// TIA Portal V20 export
TYPE "LGM_LKinCtrl_Configuration"
// stored: Access Published
   STRUCT
      referenceDesignator { ExternalAccessible := 'False'; ExternalVisible := 'False'; ExternalWritable := 'False'} : WString[25];
      disableAlarms { ExternalAccessible := 'False'; ExternalVisible := 'False'; ExternalWritable := 'False'} : Bool;
      masterControlPopUp { ExternalAccessible := 'False'; ExternalVisible := 'False'; ExternalWritable := 'False'} : Bool;
      groupPower : Struct
         startMode : Array[1.."LKINCTRL_KINEMATICS_AXES"] of DInt;   // startMode of axis; 0: enable NOT position controlled; 1: enable position controlled
         stopMode : Array[1.."LKINCTRL_KINEMATICS_AXES"] of Int;   // stopMode of axis; 0: emergency stop; 1: immediate stop; 2: stop with max dynamics
      END_STRUCT;
      groupHome : Struct
         mode : Array[1.."LKINCTRL_KINEMATICS_AXES"] of Int;   // homing modes for each axis
      END_STRUCT;
      movePath : Struct
         pathDataArray { ExternalAccessible := 'False'; ExternalVisible := 'False'; ExternalWritable := 'False'} : Array[1.."LKINCTRL_NO_OF_PATHS"] of "LKinCtrl_typePathData";
         pointTable { ExternalAccessible := 'False'; ExternalVisible := 'False'; ExternalWritable := 'False'} : Array[1.."LKINCTRL_NO_OF_POINTS_AT_POINT_TABLE"] of "LKinCtrl_typePoint";
         setFlagNames { ExternalAccessible := 'False'; ExternalVisible := 'False'; ExternalWritable := 'False'} : Array[0.."LKINCTRL_NO_OF_LAST_SETFLAG"] of WString;
         valueFlagNames { ExternalAccessible := 'False'; ExternalVisible := 'False'; ExternalWritable := 'False'} : Array[0.."LKINCTRL_NO_OF_LAST_VALUEFLAG"] of WString;
         settings { ExternalAccessible := 'False'; ExternalVisible := 'False'; ExternalWritable := 'False'} : "LKinCtrl_typeSettings";
         pathTransition : DInt;   // initial transition configuration for new path motion (1: use bufferMode and transitionParameter)
         bufferMode : DInt := 1;   // inital bufferMode for new path motion
         transitionParameter : Array[1..5] of LReal;   // initial transitionParameter for new path motion
      END_STRUCT;
   END_STRUCT;
   // groupPower.startMode[1..6] := 1;
   // movePath.pathDataArray[1].pathDataName := 'contour';
   // movePath.pathDataArray[2].pathDataName := 'contourOCS';
   // movePath.pathDataArray[3].pathDataName := 'Packaging';
   // movePath.pathDataArray[4].pathDataName := 'PickAndPlaceTracking';
   // movePath.pathDataArray[5].pathDataName := '- - -';
   // movePath.pathDataArray[1..5].LKinLangInterface.addPointer := 0;
   // movePath.pathDataArray[1..5].LKinLangInterface.retrievePointer := 0;
   // movePath.pathDataArray[1..5].LKinLangInterface.addPointerRestarted := FALSE;
   // movePath.pathDataArray[1..5].LKinLangInterface.ignoreAddPointer := TRUE;
   // movePath.pathDataArray[1..5].LKinLangInterface.bufferLocked := FALSE;
   // movePath.pathDataArray[1..5].LKinLangInterface.preprocessingStop := FALSE;
   // movePath.pathDataArray[1].commands[1..2].cmdType := 1;
   // movePath.pathDataArray[1].commands[3].cmdType := 3;
   // movePath.pathDataArray[1].commands[4..5].cmdType := 1;
   // movePath.pathDataArray[1].commands[6].cmdType := 100;
   // movePath.pathDataArray[1].commands[7].cmdType := 3;
   // movePath.pathDataArray[1].commands[8].cmdType := 1;
   // movePath.pathDataArray[1].commands[9].cmdType := 3;
   // movePath.pathDataArray[1].commands[10].cmdType := 2;
   // movePath.pathDataArray[1].commands[11..20].cmdType := -1;
   // movePath.pathDataArray[2].commands[1].cmdType := 20;
   // movePath.pathDataArray[2].commands[2..3].cmdType := 1;
   // movePath.pathDataArray[2].commands[4].cmdType := 3;
   // movePath.pathDataArray[2].commands[5..6].cmdType := 1;
   // movePath.pathDataArray[2].commands[7].cmdType := 100;
   // movePath.pathDataArray[2].commands[8].cmdType := 3;
   // movePath.pathDataArray[2].commands[9].cmdType := 1;
   // movePath.pathDataArray[2].commands[10].cmdType := 3;
   // movePath.pathDataArray[2].commands[11].cmdType := 2;
   // movePath.pathDataArray[2].commands[12..20].cmdType := -1;
   // movePath.pathDataArray[3].commands[1..6].cmdType := 1;
   // movePath.pathDataArray[3].commands[7..20].cmdType := -1;
   // movePath.pathDataArray[4].commands[1].cmdType := 0;
   // movePath.pathDataArray[4].commands[2].cmdType := 11;
   // movePath.pathDataArray[4].commands[3].cmdType := 100;
   // movePath.pathDataArray[4].commands[4].cmdType := 11;
   // movePath.pathDataArray[4].commands[5].cmdType := 100;
   // movePath.pathDataArray[4].commands[6].cmdType := 11;
   // movePath.pathDataArray[4].commands[7..20].cmdType := -1;
   // movePath.pathDataArray[5].commands[1..20].cmdType := -1;
   // movePath.pathDataArray[1].commands[1..5].cmdActivated := TRUE;
   // movePath.pathDataArray[1].commands[6].cmdActivated := FALSE;
   // movePath.pathDataArray[1].commands[7..20].cmdActivated := TRUE;
   // movePath.pathDataArray[2].commands[1..6].cmdActivated := TRUE;
   // movePath.pathDataArray[2].commands[7].cmdActivated := FALSE;
   // movePath.pathDataArray[2].commands[8..20].cmdActivated := TRUE;
   // movePath.pathDataArray[3].commands[1..20].cmdActivated := TRUE;
   // movePath.pathDataArray[4].commands[1..20].cmdActivated := TRUE;
   // movePath.pathDataArray[5].commands[1..20].cmdActivated := TRUE;
   // movePath.pathDataArray[1].commands[1].cmdName := 'B_up';
   // movePath.pathDataArray[1].commands[2].cmdName := 'B';
   // movePath.pathDataArray[1].commands[3].cmdName := 'Circ';
   // movePath.pathDataArray[1].commands[4].cmdName := 'D_up';
   // movePath.pathDataArray[1].commands[5].cmdName := 'D';
   // movePath.pathDataArray[1].commands[6].cmdName := '';
   // movePath.pathDataArray[1].commands[7].cmdName := 'S_up';
   // movePath.pathDataArray[1].commands[8].cmdName := 'F';
   // movePath.pathDataArray[1].commands[9].cmdName := 'S_lo';
   // movePath.pathDataArray[1].commands[10].cmdName := '- - -';
   // movePath.pathDataArray[1].commands[11].cmdName := '';
   // movePath.pathDataArray[1].commands[12].cmdName := '- - -';
   // movePath.pathDataArray[1].commands[13..20].cmdName := '';
   // movePath.pathDataArray[2].commands[1].cmdName := '';
   // movePath.pathDataArray[2].commands[2].cmdName := 'B_up';
   // movePath.pathDataArray[2].commands[3].cmdName := 'B';
   // movePath.pathDataArray[2].commands[4].cmdName := 'Circ';
   // movePath.pathDataArray[2].commands[5].cmdName := 'D_up';
   // movePath.pathDataArray[2].commands[6].cmdName := 'D';
   // movePath.pathDataArray[2].commands[7].cmdName := '';
   // movePath.pathDataArray[2].commands[8].cmdName := 'S_up';
   // movePath.pathDataArray[2].commands[9].cmdName := 'F';
   // movePath.pathDataArray[2].commands[10].cmdName := 'S_lo';
   // movePath.pathDataArray[2].commands[11].cmdName := '- - -';
   // movePath.pathDataArray[2].commands[12..20].cmdName := '';
   // movePath.pathDataArray[3].commands[1..20].cmdName := '- - -';
   // movePath.pathDataArray[4].commands[1..20].cmdName := '- - -';
   // movePath.pathDataArray[5].commands[1..20].cmdName := '- - -';
   // movePath.pathDataArray[1].commands[1..20].point := -1;
   // movePath.pathDataArray[2].commands[1..20].point := -1;
   // movePath.pathDataArray[3].commands[1..3].point := -1;
   // movePath.pathDataArray[3].commands[4].point := 1;
   // movePath.pathDataArray[3].commands[5].point := 2;
   // movePath.pathDataArray[3].commands[6].point := 1;
   // movePath.pathDataArray[3].commands[7..20].point := -1;
   // movePath.pathDataArray[4].commands[1..20].point := -1;
   // movePath.pathDataArray[5].commands[1..20].point := -1;
   // movePath.pathDataArray[1].commands[1..2].measurementCmd := 0;
   // movePath.pathDataArray[1].commands[3].measurementCmd := 1;
   // movePath.pathDataArray[1].commands[4..20].measurementCmd := 0;
   // movePath.pathDataArray[2].commands[1..20].measurementCmd := 0;
   // movePath.pathDataArray[3].commands[1..20].measurementCmd := 0;
   // movePath.pathDataArray[4].commands[1..20].measurementCmd := 0;
   // movePath.pathDataArray[5].commands[1..20].measurementCmd := 0;
   // movePath.pathDataArray[1].commands[1..3].cmdCoordinates.cartesianPosition.x := 0.0;
   // movePath.pathDataArray[1].commands[4..5].cmdCoordinates.cartesianPosition.x := 10.0;
   // movePath.pathDataArray[1].commands[6..7].cmdCoordinates.cartesianPosition.x := 0.0;
   // movePath.pathDataArray[1].commands[8].cmdCoordinates.cartesianPosition.x := 5.74;
   // movePath.pathDataArray[1].commands[9..20].cmdCoordinates.cartesianPosition.x := 0.0;
   // movePath.pathDataArray[2].commands[1].cmdCoordinates.cartesianPosition.x := 100.0;
   // movePath.pathDataArray[2].commands[2..4].cmdCoordinates.cartesianPosition.x := 0.0;
   // movePath.pathDataArray[2].commands[5..6].cmdCoordinates.cartesianPosition.x := 10.0;
   // movePath.pathDataArray[2].commands[7..8].cmdCoordinates.cartesianPosition.x := 0.0;
   // movePath.pathDataArray[2].commands[9].cmdCoordinates.cartesianPosition.x := 5.74;
   // movePath.pathDataArray[2].commands[10..20].cmdCoordinates.cartesianPosition.x := 0.0;
   // movePath.pathDataArray[3].commands[1..20].cmdCoordinates.cartesianPosition.x := 0.0;
   // movePath.pathDataArray[4].commands[1..3].cmdCoordinates.cartesianPosition.x := 0.0;
   // movePath.pathDataArray[4].commands[4].cmdCoordinates.cartesianPosition.x := 50.0;
   // movePath.pathDataArray[4].commands[5].cmdCoordinates.cartesianPosition.x := 0.0;
   // movePath.pathDataArray[4].commands[6].cmdCoordinates.cartesianPosition.x := 50.0;
   // movePath.pathDataArray[4].commands[7..20].cmdCoordinates.cartesianPosition.x := 0.0;
   // movePath.pathDataArray[5].commands[1..20].cmdCoordinates.cartesianPosition.x := 0.0;
   // movePath.pathDataArray[1].commands[1..2].cmdCoordinates.cartesianPosition.y := 28.28;
   // movePath.pathDataArray[1].commands[3].cmdCoordinates.cartesianPosition.y := 0.0;
   // movePath.pathDataArray[1].commands[4..5].cmdCoordinates.cartesianPosition.y := 10.0;
   // movePath.pathDataArray[1].commands[6..7].cmdCoordinates.cartesianPosition.y := 0.0;
   // movePath.pathDataArray[1].commands[8].cmdCoordinates.cartesianPosition.y := -1.81;
   // movePath.pathDataArray[1].commands[9..20].cmdCoordinates.cartesianPosition.y := 0.0;
   // movePath.pathDataArray[2].commands[1].cmdCoordinates.cartesianPosition.y := 0.0;
   // movePath.pathDataArray[2].commands[2..3].cmdCoordinates.cartesianPosition.y := 28.28;
   // movePath.pathDataArray[2].commands[4].cmdCoordinates.cartesianPosition.y := 0.0;
   // movePath.pathDataArray[2].commands[5..6].cmdCoordinates.cartesianPosition.y := 10.0;
   // movePath.pathDataArray[2].commands[7..8].cmdCoordinates.cartesianPosition.y := 0.0;
   // movePath.pathDataArray[2].commands[9].cmdCoordinates.cartesianPosition.y := -1.81;
   // movePath.pathDataArray[2].commands[10..20].cmdCoordinates.cartesianPosition.y := 0.0;
   // movePath.pathDataArray[3].commands[1..20].cmdCoordinates.cartesianPosition.y := 0.0;
   // movePath.pathDataArray[4].commands[1..20].cmdCoordinates.cartesianPosition.y := 0.0;
   // movePath.pathDataArray[5].commands[1..20].cmdCoordinates.cartesianPosition.y := 0.0;
   // movePath.pathDataArray[1].commands[1].cmdCoordinates.cartesianPosition.z := 50.0;
   // movePath.pathDataArray[1].commands[2..3].cmdCoordinates.cartesianPosition.z := 0.0;
   // movePath.pathDataArray[1].commands[4].cmdCoordinates.cartesianPosition.z := 50.0;
   // movePath.pathDataArray[1].commands[5..9].cmdCoordinates.cartesianPosition.z := 0.0;
   // movePath.pathDataArray[1].commands[10].cmdCoordinates.cartesianPosition.z := 50.0;
   // movePath.pathDataArray[1].commands[11..20].cmdCoordinates.cartesianPosition.z := 0.0;
   // movePath.pathDataArray[2].commands[1].cmdCoordinates.cartesianPosition.z := 0.0;
   // movePath.pathDataArray[2].commands[2].cmdCoordinates.cartesianPosition.z := 50.0;
   // movePath.pathDataArray[2].commands[3..4].cmdCoordinates.cartesianPosition.z := 0.0;
   // movePath.pathDataArray[2].commands[5].cmdCoordinates.cartesianPosition.z := 50.0;
   // movePath.pathDataArray[2].commands[6..10].cmdCoordinates.cartesianPosition.z := 0.0;
   // movePath.pathDataArray[2].commands[11].cmdCoordinates.cartesianPosition.z := 50.0;
   // movePath.pathDataArray[2].commands[12..20].cmdCoordinates.cartesianPosition.z := 0.0;
   // movePath.pathDataArray[3].commands[1].cmdCoordinates.cartesianPosition.z := 50.0;
   // movePath.pathDataArray[3].commands[2].cmdCoordinates.cartesianPosition.z := 10.0;
   // movePath.pathDataArray[3].commands[3].cmdCoordinates.cartesianPosition.z := 50.0;
   // movePath.pathDataArray[3].commands[4..20].cmdCoordinates.cartesianPosition.z := 0.0;
   // movePath.pathDataArray[4].commands[1].cmdCoordinates.cartesianPosition.z := 0.0;
   // movePath.pathDataArray[4].commands[2].cmdCoordinates.cartesianPosition.z := 10.0;
   // movePath.pathDataArray[4].commands[3].cmdCoordinates.cartesianPosition.z := 0.0;
   // movePath.pathDataArray[4].commands[4].cmdCoordinates.cartesianPosition.z := 10.0;
   // movePath.pathDataArray[4].commands[5].cmdCoordinates.cartesianPosition.z := 0.0;
   // movePath.pathDataArray[4].commands[6].cmdCoordinates.cartesianPosition.z := 80.0;
   // movePath.pathDataArray[4].commands[7..20].cmdCoordinates.cartesianPosition.z := 0.0;
   // movePath.pathDataArray[5].commands[1..20].cmdCoordinates.cartesianPosition.z := 0.0;
   // movePath.pathDataArray[1].commands[1..20].cmdCoordinates.cartesianPosition."a" := 0.0;
   // movePath.pathDataArray[2].commands[1..20].cmdCoordinates.cartesianPosition."a" := 0.0;
   // movePath.pathDataArray[3].commands[1..20].cmdCoordinates.cartesianPosition."a" := 0.0;
   // movePath.pathDataArray[4].commands[1..3].cmdCoordinates.cartesianPosition."a" := 0.0;
   // movePath.pathDataArray[4].commands[4].cmdCoordinates.cartesianPosition."a" := 90.0;
   // movePath.pathDataArray[4].commands[5..20].cmdCoordinates.cartesianPosition."a" := 0.0;
   // movePath.pathDataArray[5].commands[1..20].cmdCoordinates.cartesianPosition."a" := 0.0;
   // movePath.pathDataArray[1].commands[1..20].cmdCoordinates.cartesianPosition."b" := 0.0;
   // movePath.pathDataArray[2].commands[1..20].cmdCoordinates.cartesianPosition."b" := 0.0;
   // movePath.pathDataArray[3].commands[1..20].cmdCoordinates.cartesianPosition."b" := 0.0;
   // movePath.pathDataArray[4].commands[1..20].cmdCoordinates.cartesianPosition."b" := 0.0;
   // movePath.pathDataArray[5].commands[1..20].cmdCoordinates.cartesianPosition."b" := 0.0;
   // movePath.pathDataArray[1].commands[1..20].cmdCoordinates.cartesianPosition.c := 0.0;
   // movePath.pathDataArray[2].commands[1..20].cmdCoordinates.cartesianPosition.c := 0.0;
   // movePath.pathDataArray[3].commands[1..20].cmdCoordinates.cartesianPosition.c := 0.0;
   // movePath.pathDataArray[4].commands[1..20].cmdCoordinates.cartesianPosition.c := 0.0;
   // movePath.pathDataArray[5].commands[1..20].cmdCoordinates.cartesianPosition.c := 0.0;
   // movePath.pathDataArray[1].commands[1..20].cmdCoordinates.coordSystem := 0;
   // movePath.pathDataArray[2].commands[1..6].cmdCoordinates.coordSystem := 3;
   // movePath.pathDataArray[2].commands[7].cmdCoordinates.coordSystem := 0;
   // movePath.pathDataArray[2].commands[8..10].cmdCoordinates.coordSystem := 3;
   // movePath.pathDataArray[2].commands[11..20].cmdCoordinates.coordSystem := 0;
   // movePath.pathDataArray[3].commands[1..20].cmdCoordinates.coordSystem := 0;
   // movePath.pathDataArray[4].commands[1].cmdCoordinates.coordSystem := 0;
   // movePath.pathDataArray[4].commands[2].cmdCoordinates.coordSystem := 1;
   // movePath.pathDataArray[4].commands[3].cmdCoordinates.coordSystem := 0;
   // movePath.pathDataArray[4].commands[4].cmdCoordinates.coordSystem := 2;
   // movePath.pathDataArray[4].commands[5..20].cmdCoordinates.coordSystem := 0;
   // movePath.pathDataArray[5].commands[1..20].cmdCoordinates.coordSystem := 0;
   // movePath.pathDataArray[1].commands[1..2].cmdParameters.pathDynamics.velocity := 300.0;
   // movePath.pathDataArray[1].commands[3].cmdParameters.pathDynamics.velocity := 150.0;
   // movePath.pathDataArray[1].commands[4..5].cmdParameters.pathDynamics.velocity := 300.0;
   // movePath.pathDataArray[1].commands[6].cmdParameters.pathDynamics.velocity := 3000.0;
   // movePath.pathDataArray[1].commands[7].cmdParameters.pathDynamics.velocity := 150.0;
   // movePath.pathDataArray[1].commands[8].cmdParameters.pathDynamics.velocity := 300.0;
   // movePath.pathDataArray[1].commands[9].cmdParameters.pathDynamics.velocity := 150.0;
   // movePath.pathDataArray[1].commands[10..20].cmdParameters.pathDynamics.velocity := -1.0;
   // movePath.pathDataArray[2].commands[1].cmdParameters.pathDynamics.velocity := -1.0;
   // movePath.pathDataArray[2].commands[2..3].cmdParameters.pathDynamics.velocity := 300.0;
   // movePath.pathDataArray[2].commands[4].cmdParameters.pathDynamics.velocity := 150.0;
   // movePath.pathDataArray[2].commands[5..6].cmdParameters.pathDynamics.velocity := 300.0;
   // movePath.pathDataArray[2].commands[7].cmdParameters.pathDynamics.velocity := 3000.0;
   // movePath.pathDataArray[2].commands[8].cmdParameters.pathDynamics.velocity := 150.0;
   // movePath.pathDataArray[2].commands[9].cmdParameters.pathDynamics.velocity := 300.0;
   // movePath.pathDataArray[2].commands[10].cmdParameters.pathDynamics.velocity := 150.0;
   // movePath.pathDataArray[2].commands[11..20].cmdParameters.pathDynamics.velocity := -1.0;
   // movePath.pathDataArray[3].commands[1..20].cmdParameters.pathDynamics.velocity := -1.0;
   // movePath.pathDataArray[4].commands[1].cmdParameters.pathDynamics.velocity := -1.0;
   // movePath.pathDataArray[4].commands[2..6].cmdParameters.pathDynamics.velocity := 200.0;
   // movePath.pathDataArray[4].commands[7..20].cmdParameters.pathDynamics.velocity := -1.0;
   // movePath.pathDataArray[5].commands[1..20].cmdParameters.pathDynamics.velocity := -1.0;
   // movePath.pathDataArray[1].commands[1..20].cmdParameters.pathDynamics.acceleration := -1.0;
   // movePath.pathDataArray[2].commands[1..20].cmdParameters.pathDynamics.acceleration := -1.0;
   // movePath.pathDataArray[3].commands[1..20].cmdParameters.pathDynamics.acceleration := -1.0;
   // movePath.pathDataArray[4].commands[1..20].cmdParameters.pathDynamics.acceleration := -1.0;
   // movePath.pathDataArray[5].commands[1..20].cmdParameters.pathDynamics.acceleration := -1.0;
   // movePath.pathDataArray[1].commands[1..20].cmdParameters.pathDynamics.deceleration := -1.0;
   // movePath.pathDataArray[2].commands[1..20].cmdParameters.pathDynamics.deceleration := -1.0;
   // movePath.pathDataArray[3].commands[1..20].cmdParameters.pathDynamics.deceleration := -1.0;
   // movePath.pathDataArray[4].commands[1..20].cmdParameters.pathDynamics.deceleration := -1.0;
   // movePath.pathDataArray[5].commands[1..20].cmdParameters.pathDynamics.deceleration := -1.0;
   // movePath.pathDataArray[1].commands[1..20].cmdParameters.pathDynamics.jerk := -1.0;
   // movePath.pathDataArray[2].commands[1..20].cmdParameters.pathDynamics.jerk := -1.0;
   // movePath.pathDataArray[3].commands[1..20].cmdParameters.pathDynamics.jerk := -1.0;
   // movePath.pathDataArray[4].commands[1..20].cmdParameters.pathDynamics.jerk := -1.0;
   // movePath.pathDataArray[5].commands[1..20].cmdParameters.pathDynamics.jerk := -1.0;
   // movePath.pathDataArray[1].commands[1..20].cmdParameters.orientationDynamics.velocity := -1.0;
   // movePath.pathDataArray[2].commands[1..20].cmdParameters.orientationDynamics.velocity := -1.0;
   // movePath.pathDataArray[3].commands[1..20].cmdParameters.orientationDynamics.velocity := -1.0;
   // movePath.pathDataArray[4].commands[1..20].cmdParameters.orientationDynamics.velocity := -1.0;
   // movePath.pathDataArray[5].commands[1..20].cmdParameters.orientationDynamics.velocity := -1.0;
   // movePath.pathDataArray[1].commands[1..20].cmdParameters.orientationDynamics.acceleration := -1.0;
   // movePath.pathDataArray[2].commands[1..20].cmdParameters.orientationDynamics.acceleration := -1.0;
   // movePath.pathDataArray[3].commands[1..20].cmdParameters.orientationDynamics.acceleration := -1.0;
   // movePath.pathDataArray[4].commands[1..20].cmdParameters.orientationDynamics.acceleration := -1.0;
   // movePath.pathDataArray[5].commands[1..20].cmdParameters.orientationDynamics.acceleration := -1.0;
   // movePath.pathDataArray[1].commands[1..20].cmdParameters.orientationDynamics.deceleration := -1.0;
   // movePath.pathDataArray[2].commands[1..20].cmdParameters.orientationDynamics.deceleration := -1.0;
   // movePath.pathDataArray[3].commands[1..20].cmdParameters.orientationDynamics.deceleration := -1.0;
   // movePath.pathDataArray[4].commands[1..20].cmdParameters.orientationDynamics.deceleration := -1.0;
   // movePath.pathDataArray[5].commands[1..20].cmdParameters.orientationDynamics.deceleration := -1.0;
   // movePath.pathDataArray[1].commands[1..20].cmdParameters.orientationDynamics.jerk := -1.0;
   // movePath.pathDataArray[2].commands[1..20].cmdParameters.orientationDynamics.jerk := -1.0;
   // movePath.pathDataArray[3].commands[1..20].cmdParameters.orientationDynamics.jerk := -1.0;
   // movePath.pathDataArray[4].commands[1..20].cmdParameters.orientationDynamics.jerk := -1.0;
   // movePath.pathDataArray[5].commands[1..20].cmdParameters.orientationDynamics.jerk := -1.0;
   // movePath.pathDataArray[1].commands[1..20].cmdParameters.orientationDirection := 3;
   // movePath.pathDataArray[2].commands[1..20].cmdParameters.orientationDirection := 3;
   // movePath.pathDataArray[3].commands[1..20].cmdParameters.orientationDirection := 3;
   // movePath.pathDataArray[4].commands[1..20].cmdParameters.orientationDirection := 3;
   // movePath.pathDataArray[5].commands[1..20].cmdParameters.orientationDirection := 3;
   // movePath.pathDataArray[1].commands[1..2].cmdParameters.bufferMode := 2;
   // movePath.pathDataArray[1].commands[3..4].cmdParameters.bufferMode := 1;
   // movePath.pathDataArray[1].commands[5].cmdParameters.bufferMode := 2;
   // movePath.pathDataArray[1].commands[6..7].cmdParameters.bufferMode := 1;
   // movePath.pathDataArray[1].commands[8..9].cmdParameters.bufferMode := 2;
   // movePath.pathDataArray[1].commands[10..20].cmdParameters.bufferMode := 1;
   // movePath.pathDataArray[2].commands[1].cmdParameters.bufferMode := 1;
   // movePath.pathDataArray[2].commands[2..3].cmdParameters.bufferMode := 2;
   // movePath.pathDataArray[2].commands[4..5].cmdParameters.bufferMode := 1;
   // movePath.pathDataArray[2].commands[6].cmdParameters.bufferMode := 2;
   // movePath.pathDataArray[2].commands[7..8].cmdParameters.bufferMode := 1;
   // movePath.pathDataArray[2].commands[9..10].cmdParameters.bufferMode := 2;
   // movePath.pathDataArray[2].commands[11..20].cmdParameters.bufferMode := 1;
   // movePath.pathDataArray[3].commands[1..2].cmdParameters.bufferMode := 5;
   // movePath.pathDataArray[3].commands[3].cmdParameters.bufferMode := 1;
   // movePath.pathDataArray[3].commands[4..5].cmdParameters.bufferMode := 5;
   // movePath.pathDataArray[3].commands[6..20].cmdParameters.bufferMode := 1;
   // movePath.pathDataArray[4].commands[1].cmdParameters.bufferMode := 1;
   // movePath.pathDataArray[4].commands[2].cmdParameters.bufferMode := 5;
   // movePath.pathDataArray[4].commands[3..20].cmdParameters.bufferMode := 1;
   // movePath.pathDataArray[5].commands[1..20].cmdParameters.bufferMode := 1;
   // movePath.pathDataArray[1].commands[1].cmdParameters.transitionParameters[1] := -1.0;
   // movePath.pathDataArray[1].commands[1].cmdParameters.transitionParameters[2..5] := 0.0;
   // movePath.pathDataArray[1].commands[2].cmdParameters.transitionParameters[1] := -1.0;
   // movePath.pathDataArray[1].commands[2].cmdParameters.transitionParameters[2..5] := 0.0;
   // movePath.pathDataArray[1].commands[3].cmdParameters.transitionParameters[1] := -1.0;
   // movePath.pathDataArray[1].commands[3].cmdParameters.transitionParameters[2..5] := 0.0;
   // movePath.pathDataArray[1].commands[4].cmdParameters.transitionParameters[1] := -1.0;
   // movePath.pathDataArray[1].commands[4].cmdParameters.transitionParameters[2..5] := 0.0;
   // movePath.pathDataArray[1].commands[5].cmdParameters.transitionParameters[1] := -1.0;
   // movePath.pathDataArray[1].commands[5].cmdParameters.transitionParameters[2..5] := 0.0;
   // movePath.pathDataArray[1].commands[6].cmdParameters.transitionParameters[1] := -1.0;
   // movePath.pathDataArray[1].commands[6].cmdParameters.transitionParameters[2..5] := 0.0;
   // movePath.pathDataArray[1].commands[7].cmdParameters.transitionParameters[1] := -1.0;
   // movePath.pathDataArray[1].commands[7].cmdParameters.transitionParameters[2..5] := 0.0;
   // movePath.pathDataArray[1].commands[8].cmdParameters.transitionParameters[1] := -1.0;
   // movePath.pathDataArray[1].commands[8].cmdParameters.transitionParameters[2..5] := 0.0;
   // movePath.pathDataArray[1].commands[9].cmdParameters.transitionParameters[1] := -1.0;
   // movePath.pathDataArray[1].commands[9].cmdParameters.transitionParameters[2..5] := 0.0;
   // movePath.pathDataArray[1].commands[10].cmdParameters.transitionParameters[1] := -1.0;
   // movePath.pathDataArray[1].commands[10].cmdParameters.transitionParameters[2..5] := 0.0;
   // movePath.pathDataArray[1].commands[11].cmdParameters.transitionParameters[1] := -1.0;
   // movePath.pathDataArray[1].commands[11].cmdParameters.transitionParameters[2..5] := 0.0;
   // movePath.pathDataArray[1].commands[12].cmdParameters.transitionParameters[1] := -1.0;
   // movePath.pathDataArray[1].commands[12].cmdParameters.transitionParameters[2..5] := 0.0;
   // movePath.pathDataArray[1].commands[13].cmdParameters.transitionParameters[1] := -1.0;
   // movePath.pathDataArray[1].commands[13].cmdParameters.transitionParameters[2..5] := 0.0;
   // movePath.pathDataArray[1].commands[14].cmdParameters.transitionParameters[1] := -1.0;
   // movePath.pathDataArray[1].commands[14].cmdParameters.transitionParameters[2..5] := 0.0;
   // movePath.pathDataArray[1].commands[15].cmdParameters.transitionParameters[1] := -1.0;
   // movePath.pathDataArray[1].commands[15].cmdParameters.transitionParameters[2..5] := 0.0;
   // movePath.pathDataArray[1].commands[16].cmdParameters.transitionParameters[1] := -1.0;
   // movePath.pathDataArray[1].commands[16].cmdParameters.transitionParameters[2..5] := 0.0;
   // movePath.pathDataArray[1].commands[17].cmdParameters.transitionParameters[1] := -1.0;
   // movePath.pathDataArray[1].commands[17].cmdParameters.transitionParameters[2..5] := 0.0;
   // movePath.pathDataArray[1].commands[18].cmdParameters.transitionParameters[1] := -1.0;
   // movePath.pathDataArray[1].commands[18].cmdParameters.transitionParameters[2..5] := 0.0;
   // movePath.pathDataArray[1].commands[19].cmdParameters.transitionParameters[1] := -1.0;
   // movePath.pathDataArray[1].commands[19].cmdParameters.transitionParameters[2..5] := 0.0;
   // movePath.pathDataArray[1].commands[20].cmdParameters.transitionParameters[1] := -1.0;
   // movePath.pathDataArray[1].commands[20].cmdParameters.transitionParameters[2..5] := 0.0;
   // movePath.pathDataArray[2].commands[1].cmdParameters.transitionParameters[1..5] := 0.0;
   // movePath.pathDataArray[2].commands[2].cmdParameters.transitionParameters[1] := -1.0;
   // movePath.pathDataArray[2].commands[2].cmdParameters.transitionParameters[2..5] := 0.0;
   // movePath.pathDataArray[2].commands[3].cmdParameters.transitionParameters[1] := -1.0;
   // movePath.pathDataArray[2].commands[3].cmdParameters.transitionParameters[2..5] := 0.0;
   // movePath.pathDataArray[2].commands[4].cmdParameters.transitionParameters[1..5] := 0.0;
   // movePath.pathDataArray[2].commands[5].cmdParameters.transitionParameters[1..5] := 0.0;
   // movePath.pathDataArray[2].commands[6].cmdParameters.transitionParameters[1] := -1.0;
   // movePath.pathDataArray[2].commands[6].cmdParameters.transitionParameters[2..5] := 0.0;
   // movePath.pathDataArray[2].commands[7].cmdParameters.transitionParameters[1] := -1.0;
   // movePath.pathDataArray[2].commands[7].cmdParameters.transitionParameters[2..5] := 0.0;
   // movePath.pathDataArray[2].commands[8].cmdParameters.transitionParameters[1..5] := 0.0;
   // movePath.pathDataArray[2].commands[9].cmdParameters.transitionParameters[1] := -1.0;
   // movePath.pathDataArray[2].commands[9].cmdParameters.transitionParameters[2..5] := 0.0;
   // movePath.pathDataArray[2].commands[10].cmdParameters.transitionParameters[1] := -1.0;
   // movePath.pathDataArray[2].commands[10].cmdParameters.transitionParameters[2..5] := 0.0;
   // movePath.pathDataArray[2].commands[11].cmdParameters.transitionParameters[1] := -1.0;
   // movePath.pathDataArray[2].commands[11].cmdParameters.transitionParameters[2..5] := 0.0;
   // movePath.pathDataArray[2].commands[12].cmdParameters.transitionParameters[1] := -1.0;
   // movePath.pathDataArray[2].commands[12].cmdParameters.transitionParameters[2..5] := 0.0;
   // movePath.pathDataArray[2].commands[13].cmdParameters.transitionParameters[1] := -1.0;
   // movePath.pathDataArray[2].commands[13].cmdParameters.transitionParameters[2..5] := 0.0;
   // movePath.pathDataArray[2].commands[14].cmdParameters.transitionParameters[1] := -1.0;
   // movePath.pathDataArray[2].commands[14].cmdParameters.transitionParameters[2..5] := 0.0;
   // movePath.pathDataArray[2].commands[15].cmdParameters.transitionParameters[1] := -1.0;
   // movePath.pathDataArray[2].commands[15].cmdParameters.transitionParameters[2..5] := 0.0;
   // movePath.pathDataArray[2].commands[16].cmdParameters.transitionParameters[1] := -1.0;
   // movePath.pathDataArray[2].commands[16].cmdParameters.transitionParameters[2..5] := 0.0;
   // movePath.pathDataArray[2].commands[17].cmdParameters.transitionParameters[1] := -1.0;
   // movePath.pathDataArray[2].commands[17].cmdParameters.transitionParameters[2..5] := 0.0;
   // movePath.pathDataArray[2].commands[18].cmdParameters.transitionParameters[1] := -1.0;
   // movePath.pathDataArray[2].commands[18].cmdParameters.transitionParameters[2..5] := 0.0;
   // movePath.pathDataArray[2].commands[19].cmdParameters.transitionParameters[1] := -1.0;
   // movePath.pathDataArray[2].commands[19].cmdParameters.transitionParameters[2..5] := 0.0;
   // movePath.pathDataArray[2].commands[20].cmdParameters.transitionParameters[1] := -1.0;
   // movePath.pathDataArray[2].commands[20].cmdParameters.transitionParameters[2..5] := 0.0;
   // movePath.pathDataArray[3].commands[1].cmdParameters.transitionParameters[1] := -1.0;
   // movePath.pathDataArray[3].commands[1].cmdParameters.transitionParameters[2..5] := 0.0;
   // movePath.pathDataArray[3].commands[2].cmdParameters.transitionParameters[1] := -1.0;
   // movePath.pathDataArray[3].commands[2].cmdParameters.transitionParameters[2..5] := 0.0;
   // movePath.pathDataArray[3].commands[3].cmdParameters.transitionParameters[1] := -1.0;
   // movePath.pathDataArray[3].commands[3].cmdParameters.transitionParameters[2..5] := 0.0;
   // movePath.pathDataArray[3].commands[4].cmdParameters.transitionParameters[1] := -1.0;
   // movePath.pathDataArray[3].commands[4].cmdParameters.transitionParameters[2..5] := 0.0;
   // movePath.pathDataArray[3].commands[5].cmdParameters.transitionParameters[1] := -1.0;
   // movePath.pathDataArray[3].commands[5].cmdParameters.transitionParameters[2..5] := 0.0;
   // movePath.pathDataArray[3].commands[6].cmdParameters.transitionParameters[1] := -1.0;
   // movePath.pathDataArray[3].commands[6].cmdParameters.transitionParameters[2..5] := 0.0;
   // movePath.pathDataArray[3].commands[7].cmdParameters.transitionParameters[1] := -1.0;
   // movePath.pathDataArray[3].commands[7].cmdParameters.transitionParameters[2..5] := 0.0;
   // movePath.pathDataArray[3].commands[8].cmdParameters.transitionParameters[1] := -1.0;
   // movePath.pathDataArray[3].commands[8].cmdParameters.transitionParameters[2..5] := 0.0;
   // movePath.pathDataArray[3].commands[9].cmdParameters.transitionParameters[1] := -1.0;
   // movePath.pathDataArray[3].commands[9].cmdParameters.transitionParameters[2..5] := 0.0;
   // movePath.pathDataArray[3].commands[10].cmdParameters.transitionParameters[1] := -1.0;
   // movePath.pathDataArray[3].commands[10].cmdParameters.transitionParameters[2..5] := 0.0;
   // movePath.pathDataArray[3].commands[11].cmdParameters.transitionParameters[1] := -1.0;
   // movePath.pathDataArray[3].commands[11].cmdParameters.transitionParameters[2..5] := 0.0;
   // movePath.pathDataArray[3].commands[12].cmdParameters.transitionParameters[1] := -1.0;
   // movePath.pathDataArray[3].commands[12].cmdParameters.transitionParameters[2..5] := 0.0;
   // movePath.pathDataArray[3].commands[13].cmdParameters.transitionParameters[1] := -1.0;
   // movePath.pathDataArray[3].commands[13].cmdParameters.transitionParameters[2..5] := 0.0;
   // movePath.pathDataArray[3].commands[14].cmdParameters.transitionParameters[1] := -1.0;
   // movePath.pathDataArray[3].commands[14].cmdParameters.transitionParameters[2..5] := 0.0;
   // movePath.pathDataArray[3].commands[15].cmdParameters.transitionParameters[1] := -1.0;
   // movePath.pathDataArray[3].commands[15].cmdParameters.transitionParameters[2..5] := 0.0;
   // movePath.pathDataArray[3].commands[16].cmdParameters.transitionParameters[1] := -1.0;
   // movePath.pathDataArray[3].commands[16].cmdParameters.transitionParameters[2..5] := 0.0;
   // movePath.pathDataArray[3].commands[17].cmdParameters.transitionParameters[1] := -1.0;
   // movePath.pathDataArray[3].commands[17].cmdParameters.transitionParameters[2..5] := 0.0;
   // movePath.pathDataArray[3].commands[18].cmdParameters.transitionParameters[1] := -1.0;
   // movePath.pathDataArray[3].commands[18].cmdParameters.transitionParameters[2..5] := 0.0;
   // movePath.pathDataArray[3].commands[19].cmdParameters.transitionParameters[1] := -1.0;
   // movePath.pathDataArray[3].commands[19].cmdParameters.transitionParameters[2..5] := 0.0;
   // movePath.pathDataArray[3].commands[20].cmdParameters.transitionParameters[1] := -1.0;
   // movePath.pathDataArray[3].commands[20].cmdParameters.transitionParameters[2..5] := 0.0;
   // movePath.pathDataArray[4].commands[1].cmdParameters.transitionParameters[1] := -1.0;
   // movePath.pathDataArray[4].commands[1].cmdParameters.transitionParameters[2..5] := 0.0;
   // movePath.pathDataArray[4].commands[2].cmdParameters.transitionParameters[1] := 30.0;
   // movePath.pathDataArray[4].commands[2].cmdParameters.transitionParameters[2..5] := 0.0;
   // movePath.pathDataArray[4].commands[3].cmdParameters.transitionParameters[1] := -1.0;
   // movePath.pathDataArray[4].commands[3].cmdParameters.transitionParameters[2..5] := 0.0;
   // movePath.pathDataArray[4].commands[4].cmdParameters.transitionParameters[1] := -1.0;
   // movePath.pathDataArray[4].commands[4].cmdParameters.transitionParameters[2..5] := 0.0;
   // movePath.pathDataArray[4].commands[5].cmdParameters.transitionParameters[1] := -1.0;
   // movePath.pathDataArray[4].commands[5].cmdParameters.transitionParameters[2..5] := 0.0;
   // movePath.pathDataArray[4].commands[6].cmdParameters.transitionParameters[1] := -1.0;
   // movePath.pathDataArray[4].commands[6].cmdParameters.transitionParameters[2..5] := 0.0;
   // movePath.pathDataArray[4].commands[7].cmdParameters.transitionParameters[1] := -1.0;
   // movePath.pathDataArray[4].commands[7].cmdParameters.transitionParameters[2..5] := 0.0;
   // movePath.pathDataArray[4].commands[8].cmdParameters.transitionParameters[1] := -1.0;
   // movePath.pathDataArray[4].commands[8].cmdParameters.transitionParameters[2..5] := 0.0;
   // movePath.pathDataArray[4].commands[9].cmdParameters.transitionParameters[1] := -1.0;
   // movePath.pathDataArray[4].commands[9].cmdParameters.transitionParameters[2..5] := 0.0;
   // movePath.pathDataArray[4].commands[10].cmdParameters.transitionParameters[1] := -1.0;
   // movePath.pathDataArray[4].commands[10].cmdParameters.transitionParameters[2..5] := 0.0;
   // movePath.pathDataArray[4].commands[11].cmdParameters.transitionParameters[1] := -1.0;
   // movePath.pathDataArray[4].commands[11].cmdParameters.transitionParameters[2..5] := 0.0;
   // movePath.pathDataArray[4].commands[12].cmdParameters.transitionParameters[1] := -1.0;
   // movePath.pathDataArray[4].commands[12].cmdParameters.transitionParameters[2..5] := 0.0;
   // movePath.pathDataArray[4].commands[13].cmdParameters.transitionParameters[1] := -1.0;
   // movePath.pathDataArray[4].commands[13].cmdParameters.transitionParameters[2..5] := 0.0;
   // movePath.pathDataArray[4].commands[14].cmdParameters.transitionParameters[1] := -1.0;
   // movePath.pathDataArray[4].commands[14].cmdParameters.transitionParameters[2..5] := 0.0;
   // movePath.pathDataArray[4].commands[15].cmdParameters.transitionParameters[1] := -1.0;
   // movePath.pathDataArray[4].commands[15].cmdParameters.transitionParameters[2..5] := 0.0;
   // movePath.pathDataArray[4].commands[16].cmdParameters.transitionParameters[1] := -1.0;
   // movePath.pathDataArray[4].commands[16].cmdParameters.transitionParameters[2..5] := 0.0;
   // movePath.pathDataArray[4].commands[17].cmdParameters.transitionParameters[1] := -1.0;
   // movePath.pathDataArray[4].commands[17].cmdParameters.transitionParameters[2..5] := 0.0;
   // movePath.pathDataArray[4].commands[18].cmdParameters.transitionParameters[1] := -1.0;
   // movePath.pathDataArray[4].commands[18].cmdParameters.transitionParameters[2..5] := 0.0;
   // movePath.pathDataArray[4].commands[19].cmdParameters.transitionParameters[1] := -1.0;
   // movePath.pathDataArray[4].commands[19].cmdParameters.transitionParameters[2..5] := 0.0;
   // movePath.pathDataArray[4].commands[20].cmdParameters.transitionParameters[1] := -1.0;
   // movePath.pathDataArray[4].commands[20].cmdParameters.transitionParameters[2..5] := 0.0;
   // movePath.pathDataArray[5].commands[1].cmdParameters.transitionParameters[1] := -1.0;
   // movePath.pathDataArray[5].commands[1].cmdParameters.transitionParameters[2..5] := 0.0;
   // movePath.pathDataArray[5].commands[2].cmdParameters.transitionParameters[1] := -1.0;
   // movePath.pathDataArray[5].commands[2].cmdParameters.transitionParameters[2..5] := 0.0;
   // movePath.pathDataArray[5].commands[3].cmdParameters.transitionParameters[1] := -1.0;
   // movePath.pathDataArray[5].commands[3].cmdParameters.transitionParameters[2..5] := 0.0;
   // movePath.pathDataArray[5].commands[4].cmdParameters.transitionParameters[1] := -1.0;
   // movePath.pathDataArray[5].commands[4].cmdParameters.transitionParameters[2..5] := 0.0;
   // movePath.pathDataArray[5].commands[5].cmdParameters.transitionParameters[1] := -1.0;
   // movePath.pathDataArray[5].commands[5].cmdParameters.transitionParameters[2..5] := 0.0;
   // movePath.pathDataArray[5].commands[6].cmdParameters.transitionParameters[1] := -1.0;
   // movePath.pathDataArray[5].commands[6].cmdParameters.transitionParameters[2..5] := 0.0;
   // movePath.pathDataArray[5].commands[7].cmdParameters.transitionParameters[1] := -1.0;
   // movePath.pathDataArray[5].commands[7].cmdParameters.transitionParameters[2..5] := 0.0;
   // movePath.pathDataArray[5].commands[8].cmdParameters.transitionParameters[1] := -1.0;
   // movePath.pathDataArray[5].commands[8].cmdParameters.transitionParameters[2..5] := 0.0;
   // movePath.pathDataArray[5].commands[9].cmdParameters.transitionParameters[1] := -1.0;
   // movePath.pathDataArray[5].commands[9].cmdParameters.transitionParameters[2..5] := 0.0;
   // movePath.pathDataArray[5].commands[10].cmdParameters.transitionParameters[1] := -1.0;
   // movePath.pathDataArray[5].commands[10].cmdParameters.transitionParameters[2..5] := 0.0;
   // movePath.pathDataArray[5].commands[11].cmdParameters.transitionParameters[1] := -1.0;
   // movePath.pathDataArray[5].commands[11].cmdParameters.transitionParameters[2..5] := 0.0;
   // movePath.pathDataArray[5].commands[12].cmdParameters.transitionParameters[1] := -1.0;
   // movePath.pathDataArray[5].commands[12].cmdParameters.transitionParameters[2..5] := 0.0;
   // movePath.pathDataArray[5].commands[13].cmdParameters.transitionParameters[1] := -1.0;
   // movePath.pathDataArray[5].commands[13].cmdParameters.transitionParameters[2..5] := 0.0;
   // movePath.pathDataArray[5].commands[14].cmdParameters.transitionParameters[1] := -1.0;
   // movePath.pathDataArray[5].commands[14].cmdParameters.transitionParameters[2..5] := 0.0;
   // movePath.pathDataArray[5].commands[15].cmdParameters.transitionParameters[1] := -1.0;
   // movePath.pathDataArray[5].commands[15].cmdParameters.transitionParameters[2..5] := 0.0;
   // movePath.pathDataArray[5].commands[16].cmdParameters.transitionParameters[1] := -1.0;
   // movePath.pathDataArray[5].commands[16].cmdParameters.transitionParameters[2..5] := 0.0;
   // movePath.pathDataArray[5].commands[17].cmdParameters.transitionParameters[1] := -1.0;
   // movePath.pathDataArray[5].commands[17].cmdParameters.transitionParameters[2..5] := 0.0;
   // movePath.pathDataArray[5].commands[18].cmdParameters.transitionParameters[1] := -1.0;
   // movePath.pathDataArray[5].commands[18].cmdParameters.transitionParameters[2..5] := 0.0;
   // movePath.pathDataArray[5].commands[19].cmdParameters.transitionParameters[1] := -1.0;
   // movePath.pathDataArray[5].commands[19].cmdParameters.transitionParameters[2..5] := 0.0;
   // movePath.pathDataArray[5].commands[20].cmdParameters.transitionParameters[1] := -1.0;
   // movePath.pathDataArray[5].commands[20].cmdParameters.transitionParameters[2..5] := 0.0;
   // movePath.pathDataArray[1].commands[1..20].cmdParameters.dynamicAdaption := -1;
   // movePath.pathDataArray[2].commands[1..20].cmdParameters.dynamicAdaption := -1;
   // movePath.pathDataArray[3].commands[1..20].cmdParameters.dynamicAdaption := -1;
   // movePath.pathDataArray[4].commands[1].cmdParameters.dynamicAdaption := -1;
   // movePath.pathDataArray[4].commands[2].cmdParameters.dynamicAdaption := 0;
   // movePath.pathDataArray[4].commands[3].cmdParameters.dynamicAdaption := -1;
   // movePath.pathDataArray[4].commands[4].cmdParameters.dynamicAdaption := 0;
   // movePath.pathDataArray[4].commands[5].cmdParameters.dynamicAdaption := -1;
   // movePath.pathDataArray[4].commands[6].cmdParameters.dynamicAdaption := 0;
   // movePath.pathDataArray[4].commands[7..20].cmdParameters.dynamicAdaption := -1;
   // movePath.pathDataArray[5].commands[1..20].cmdParameters.dynamicAdaption := -1;
   // movePath.pathDataArray[1].commands[1..20].cmdParameters.toolNumber := 0;
   // movePath.pathDataArray[2].commands[1..20].cmdParameters.toolNumber := 0;
   // movePath.pathDataArray[3].commands[1..20].cmdParameters.toolNumber := 0;
   // movePath.pathDataArray[4].commands[1..20].cmdParameters.toolNumber := 0;
   // movePath.pathDataArray[5].commands[1..20].cmdParameters.toolNumber := 0;
   // movePath.pathDataArray[1].commands[1..20].cmdParameters.moveDirectParameters.linkConstellation := 16#FFFF_FFFF;
   // movePath.pathDataArray[2].commands[1..20].cmdParameters.moveDirectParameters.linkConstellation := 16#FFFF_FFFF;
   // movePath.pathDataArray[3].commands[1..20].cmdParameters.moveDirectParameters.linkConstellation := 16#FFFF_FFFF;
   // movePath.pathDataArray[4].commands[1..20].cmdParameters.moveDirectParameters.linkConstellation := 16#FFFF_FFFF;
   // movePath.pathDataArray[5].commands[1..20].cmdParameters.moveDirectParameters.linkConstellation := 16#FFFF_FFFF;
   // movePath.pathDataArray[1].commands[1..20].cmdParameters.moveDirectParameters.positionMode := 1;
   // movePath.pathDataArray[2].commands[1..20].cmdParameters.moveDirectParameters.positionMode := 1;
   // movePath.pathDataArray[3].commands[1..20].cmdParameters.moveDirectParameters.positionMode := 1;
   // movePath.pathDataArray[4].commands[1..20].cmdParameters.moveDirectParameters.positionMode := 1;
   // movePath.pathDataArray[5].commands[1..20].cmdParameters.moveDirectParameters.positionMode := 1;
   // movePath.pathDataArray[1].commands[1].cmdParameters.moveDirectParameters.turnJoint[1..6] := 0;
   // movePath.pathDataArray[1].commands[2].cmdParameters.moveDirectParameters.turnJoint[1..6] := 0;
   // movePath.pathDataArray[1].commands[3].cmdParameters.moveDirectParameters.turnJoint[1..6] := 0;
   // movePath.pathDataArray[1].commands[4].cmdParameters.moveDirectParameters.turnJoint[1..6] := 0;
   // movePath.pathDataArray[1].commands[5].cmdParameters.moveDirectParameters.turnJoint[1..6] := 0;
   // movePath.pathDataArray[1].commands[6].cmdParameters.moveDirectParameters.turnJoint[1..6] := 0;
   // movePath.pathDataArray[1].commands[7].cmdParameters.moveDirectParameters.turnJoint[1..6] := 0;
   // movePath.pathDataArray[1].commands[8].cmdParameters.moveDirectParameters.turnJoint[1..6] := 0;
   // movePath.pathDataArray[1].commands[9].cmdParameters.moveDirectParameters.turnJoint[1..6] := 0;
   // movePath.pathDataArray[1].commands[10].cmdParameters.moveDirectParameters.turnJoint[1..6] := 0;
   // movePath.pathDataArray[1].commands[11].cmdParameters.moveDirectParameters.turnJoint[1..6] := 0;
   // movePath.pathDataArray[1].commands[12].cmdParameters.moveDirectParameters.turnJoint[1..6] := 0;
   // movePath.pathDataArray[1].commands[13].cmdParameters.moveDirectParameters.turnJoint[1..6] := 0;
   // movePath.pathDataArray[1].commands[14].cmdParameters.moveDirectParameters.turnJoint[1..6] := 0;
   // movePath.pathDataArray[1].commands[15].cmdParameters.moveDirectParameters.turnJoint[1..6] := 0;
   // movePath.pathDataArray[1].commands[16].cmdParameters.moveDirectParameters.turnJoint[1..6] := 0;
   // movePath.pathDataArray[1].commands[17].cmdParameters.moveDirectParameters.turnJoint[1..6] := 0;
   // movePath.pathDataArray[1].commands[18].cmdParameters.moveDirectParameters.turnJoint[1..6] := 0;
   // movePath.pathDataArray[1].commands[19].cmdParameters.moveDirectParameters.turnJoint[1..6] := 0;
   // movePath.pathDataArray[1].commands[20].cmdParameters.moveDirectParameters.turnJoint[1..6] := 0;
   // movePath.pathDataArray[2].commands[1].cmdParameters.moveDirectParameters.turnJoint[1..6] := 0;
   // movePath.pathDataArray[2].commands[2].cmdParameters.moveDirectParameters.turnJoint[1..6] := 0;
   // movePath.pathDataArray[2].commands[3].cmdParameters.moveDirectParameters.turnJoint[1..6] := 0;
   // movePath.pathDataArray[2].commands[4].cmdParameters.moveDirectParameters.turnJoint[1..6] := 0;
   // movePath.pathDataArray[2].commands[5].cmdParameters.moveDirectParameters.turnJoint[1..6] := 0;
   // movePath.pathDataArray[2].commands[6].cmdParameters.moveDirectParameters.turnJoint[1..6] := 0;
   // movePath.pathDataArray[2].commands[7].cmdParameters.moveDirectParameters.turnJoint[1..6] := 0;
   // movePath.pathDataArray[2].commands[8].cmdParameters.moveDirectParameters.turnJoint[1..6] := 0;
   // movePath.pathDataArray[2].commands[9].cmdParameters.moveDirectParameters.turnJoint[1..6] := 0;
   // movePath.pathDataArray[2].commands[10].cmdParameters.moveDirectParameters.turnJoint[1..6] := 0;
   // movePath.pathDataArray[2].commands[11].cmdParameters.moveDirectParameters.turnJoint[1..6] := 0;
   // movePath.pathDataArray[2].commands[12].cmdParameters.moveDirectParameters.turnJoint[1..6] := 0;
   // movePath.pathDataArray[2].commands[13].cmdParameters.moveDirectParameters.turnJoint[1..6] := 0;
   // movePath.pathDataArray[2].commands[14].cmdParameters.moveDirectParameters.turnJoint[1..6] := 0;
   // movePath.pathDataArray[2].commands[15].cmdParameters.moveDirectParameters.turnJoint[1..6] := 0;
   // movePath.pathDataArray[2].commands[16].cmdParameters.moveDirectParameters.turnJoint[1..6] := 0;
   // movePath.pathDataArray[2].commands[17].cmdParameters.moveDirectParameters.turnJoint[1..6] := 0;
   // movePath.pathDataArray[2].commands[18].cmdParameters.moveDirectParameters.turnJoint[1..6] := 0;
   // movePath.pathDataArray[2].commands[19].cmdParameters.moveDirectParameters.turnJoint[1..6] := 0;
   // movePath.pathDataArray[2].commands[20].cmdParameters.moveDirectParameters.turnJoint[1..6] := 0;
   // movePath.pathDataArray[3].commands[1].cmdParameters.moveDirectParameters.turnJoint[1..6] := 0;
   // movePath.pathDataArray[3].commands[2].cmdParameters.moveDirectParameters.turnJoint[1..6] := 0;
   // movePath.pathDataArray[3].commands[3].cmdParameters.moveDirectParameters.turnJoint[1..6] := 0;
   // movePath.pathDataArray[3].commands[4].cmdParameters.moveDirectParameters.turnJoint[1..6] := 0;
   // movePath.pathDataArray[3].commands[5].cmdParameters.moveDirectParameters.turnJoint[1..6] := 0;
   // movePath.pathDataArray[3].commands[6].cmdParameters.moveDirectParameters.turnJoint[1..6] := 0;
   // movePath.pathDataArray[3].commands[7].cmdParameters.moveDirectParameters.turnJoint[1..6] := 0;
   // movePath.pathDataArray[3].commands[8].cmdParameters.moveDirectParameters.turnJoint[1..6] := 0;
   // movePath.pathDataArray[3].commands[9].cmdParameters.moveDirectParameters.turnJoint[1..6] := 0;
   // movePath.pathDataArray[3].commands[10].cmdParameters.moveDirectParameters.turnJoint[1..6] := 0;
   // movePath.pathDataArray[3].commands[11].cmdParameters.moveDirectParameters.turnJoint[1..6] := 0;
   // movePath.pathDataArray[3].commands[12].cmdParameters.moveDirectParameters.turnJoint[1..6] := 0;
   // movePath.pathDataArray[3].commands[13].cmdParameters.moveDirectParameters.turnJoint[1..6] := 0;
   // movePath.pathDataArray[3].commands[14].cmdParameters.moveDirectParameters.turnJoint[1..6] := 0;
   // movePath.pathDataArray[3].commands[15].cmdParameters.moveDirectParameters.turnJoint[1..6] := 0;
   // movePath.pathDataArray[3].commands[16].cmdParameters.moveDirectParameters.turnJoint[1..6] := 0;
   // movePath.pathDataArray[3].commands[17].cmdParameters.moveDirectParameters.turnJoint[1..6] := 0;
   // movePath.pathDataArray[3].commands[18].cmdParameters.moveDirectParameters.turnJoint[1..6] := 0;
   // movePath.pathDataArray[3].commands[19].cmdParameters.moveDirectParameters.turnJoint[1..6] := 0;
   // movePath.pathDataArray[3].commands[20].cmdParameters.moveDirectParameters.turnJoint[1..6] := 0;
   // movePath.pathDataArray[4].commands[1].cmdParameters.moveDirectParameters.turnJoint[1..6] := 0;
   // movePath.pathDataArray[4].commands[2].cmdParameters.moveDirectParameters.turnJoint[1..6] := 0;
   // movePath.pathDataArray[4].commands[3].cmdParameters.moveDirectParameters.turnJoint[1..6] := 0;
   // movePath.pathDataArray[4].commands[4].cmdParameters.moveDirectParameters.turnJoint[1..6] := 0;
   // movePath.pathDataArray[4].commands[5].cmdParameters.moveDirectParameters.turnJoint[1..6] := 0;
   // movePath.pathDataArray[4].commands[6].cmdParameters.moveDirectParameters.turnJoint[1..6] := 0;
   // movePath.pathDataArray[4].commands[7].cmdParameters.moveDirectParameters.turnJoint[1..6] := 0;
   // movePath.pathDataArray[4].commands[8].cmdParameters.moveDirectParameters.turnJoint[1..6] := 0;
   // movePath.pathDataArray[4].commands[9].cmdParameters.moveDirectParameters.turnJoint[1..6] := 0;
   // movePath.pathDataArray[4].commands[10].cmdParameters.moveDirectParameters.turnJoint[1..6] := 0;
   // movePath.pathDataArray[4].commands[11].cmdParameters.moveDirectParameters.turnJoint[1..6] := 0;
   // movePath.pathDataArray[4].commands[12].cmdParameters.moveDirectParameters.turnJoint[1..6] := 0;
   // movePath.pathDataArray[4].commands[13].cmdParameters.moveDirectParameters.turnJoint[1..6] := 0;
   // movePath.pathDataArray[4].commands[14].cmdParameters.moveDirectParameters.turnJoint[1..6] := 0;
   // movePath.pathDataArray[4].commands[15].cmdParameters.moveDirectParameters.turnJoint[1..6] := 0;
   // movePath.pathDataArray[4].commands[16].cmdParameters.moveDirectParameters.turnJoint[1..6] := 0;
   // movePath.pathDataArray[4].commands[17].cmdParameters.moveDirectParameters.turnJoint[1..6] := 0;
   // movePath.pathDataArray[4].commands[18].cmdParameters.moveDirectParameters.turnJoint[1..6] := 0;
   // movePath.pathDataArray[4].commands[19].cmdParameters.moveDirectParameters.turnJoint[1..6] := 0;
   // movePath.pathDataArray[4].commands[20].cmdParameters.moveDirectParameters.turnJoint[1..6] := 0;
   // movePath.pathDataArray[5].commands[1].cmdParameters.moveDirectParameters.turnJoint[1..6] := 0;
   // movePath.pathDataArray[5].commands[2].cmdParameters.moveDirectParameters.turnJoint[1..6] := 0;
   // movePath.pathDataArray[5].commands[3].cmdParameters.moveDirectParameters.turnJoint[1..6] := 0;
   // movePath.pathDataArray[5].commands[4].cmdParameters.moveDirectParameters.turnJoint[1..6] := 0;
   // movePath.pathDataArray[5].commands[5].cmdParameters.moveDirectParameters.turnJoint[1..6] := 0;
   // movePath.pathDataArray[5].commands[6].cmdParameters.moveDirectParameters.turnJoint[1..6] := 0;
   // movePath.pathDataArray[5].commands[7].cmdParameters.moveDirectParameters.turnJoint[1..6] := 0;
   // movePath.pathDataArray[5].commands[8].cmdParameters.moveDirectParameters.turnJoint[1..6] := 0;
   // movePath.pathDataArray[5].commands[9].cmdParameters.moveDirectParameters.turnJoint[1..6] := 0;
   // movePath.pathDataArray[5].commands[10].cmdParameters.moveDirectParameters.turnJoint[1..6] := 0;
   // movePath.pathDataArray[5].commands[11].cmdParameters.moveDirectParameters.turnJoint[1..6] := 0;
   // movePath.pathDataArray[5].commands[12].cmdParameters.moveDirectParameters.turnJoint[1..6] := 0;
   // movePath.pathDataArray[5].commands[13].cmdParameters.moveDirectParameters.turnJoint[1..6] := 0;
   // movePath.pathDataArray[5].commands[14].cmdParameters.moveDirectParameters.turnJoint[1..6] := 0;
   // movePath.pathDataArray[5].commands[15].cmdParameters.moveDirectParameters.turnJoint[1..6] := 0;
   // movePath.pathDataArray[5].commands[16].cmdParameters.moveDirectParameters.turnJoint[1..6] := 0;
   // movePath.pathDataArray[5].commands[17].cmdParameters.moveDirectParameters.turnJoint[1..6] := 0;
   // movePath.pathDataArray[5].commands[18].cmdParameters.moveDirectParameters.turnJoint[1..6] := 0;
   // movePath.pathDataArray[5].commands[19].cmdParameters.moveDirectParameters.turnJoint[1..6] := 0;
   // movePath.pathDataArray[5].commands[20].cmdParameters.moveDirectParameters.turnJoint[1..6] := 0;
   // movePath.pathDataArray[1].commands[1].cmdParameters.offsetParameters.offsetParaNo := 3;
   // movePath.pathDataArray[1].commands[2..20].cmdParameters.offsetParameters.offsetParaNo := 0;
   // movePath.pathDataArray[2].commands[1].cmdParameters.offsetParameters.offsetParaNo := 1;
   // movePath.pathDataArray[2].commands[2..6].cmdParameters.offsetParameters.offsetParaNo := 3;
   // movePath.pathDataArray[2].commands[7].cmdParameters.offsetParameters.offsetParaNo := 0;
   // movePath.pathDataArray[2].commands[8..10].cmdParameters.offsetParameters.offsetParaNo := 3;
   // movePath.pathDataArray[2].commands[11..20].cmdParameters.offsetParameters.offsetParaNo := 0;
   // movePath.pathDataArray[3].commands[1..20].cmdParameters.offsetParameters.offsetParaNo := 0;
   // movePath.pathDataArray[4].commands[1..20].cmdParameters.offsetParameters.offsetParaNo := 0;
   // movePath.pathDataArray[5].commands[1..20].cmdParameters.offsetParameters.offsetParaNo := 0;
   // movePath.pathDataArray[1].commands[1..20].cmdParameters.offsetParameters.mainPathPlane := 0;
   // movePath.pathDataArray[2].commands[1..20].cmdParameters.offsetParameters.mainPathPlane := 0;
   // movePath.pathDataArray[3].commands[1..20].cmdParameters.offsetParameters.mainPathPlane := 0;
   // movePath.pathDataArray[4].commands[1..20].cmdParameters.offsetParameters.mainPathPlane := 0;
   // movePath.pathDataArray[5].commands[1..20].cmdParameters.offsetParameters.mainPathPlane := 0;
   // movePath.pathDataArray[1].commands[1..9].cmdParameters.conveyorParameters.conveyorParaNo := 1;
   // movePath.pathDataArray[1].commands[10].cmdParameters.conveyorParameters.conveyorParaNo := 0;
   // movePath.pathDataArray[1].commands[11].cmdParameters.conveyorParameters.conveyorParaNo := 1;
   // movePath.pathDataArray[1].commands[12].cmdParameters.conveyorParameters.conveyorParaNo := 0;
   // movePath.pathDataArray[1].commands[13..20].cmdParameters.conveyorParameters.conveyorParaNo := 1;
   // movePath.pathDataArray[2].commands[1..10].cmdParameters.conveyorParameters.conveyorParaNo := 1;
   // movePath.pathDataArray[2].commands[11].cmdParameters.conveyorParameters.conveyorParaNo := 0;
   // movePath.pathDataArray[2].commands[12..20].cmdParameters.conveyorParameters.conveyorParaNo := 1;
   // movePath.pathDataArray[3].commands[1..20].cmdParameters.conveyorParameters.conveyorParaNo := 0;
   // movePath.pathDataArray[4].commands[1].cmdParameters.conveyorParameters.conveyorParaNo := 0;
   // movePath.pathDataArray[4].commands[2].cmdParameters.conveyorParameters.conveyorParaNo := 1;
   // movePath.pathDataArray[4].commands[3].cmdParameters.conveyorParameters.conveyorParaNo := 0;
   // movePath.pathDataArray[4].commands[4].cmdParameters.conveyorParameters.conveyorParaNo := 2;
   // movePath.pathDataArray[4].commands[5..20].cmdParameters.conveyorParameters.conveyorParaNo := 0;
   // movePath.pathDataArray[5].commands[1..20].cmdParameters.conveyorParameters.conveyorParaNo := 0;
   // movePath.pathDataArray[1].commands[1..2].cmdParameters.circleParameters.circMode := 0;
   // movePath.pathDataArray[1].commands[3].cmdParameters.circleParameters.circMode := 1;
   // movePath.pathDataArray[1].commands[4..6].cmdParameters.circleParameters.circMode := 0;
   // movePath.pathDataArray[1].commands[7].cmdParameters.circleParameters.circMode := 1;
   // movePath.pathDataArray[1].commands[8].cmdParameters.circleParameters.circMode := 0;
   // movePath.pathDataArray[1].commands[9].cmdParameters.circleParameters.circMode := 1;
   // movePath.pathDataArray[1].commands[10..20].cmdParameters.circleParameters.circMode := 0;
   // movePath.pathDataArray[2].commands[1..3].cmdParameters.circleParameters.circMode := 0;
   // movePath.pathDataArray[2].commands[4].cmdParameters.circleParameters.circMode := 1;
   // movePath.pathDataArray[2].commands[5..7].cmdParameters.circleParameters.circMode := 0;
   // movePath.pathDataArray[2].commands[8].cmdParameters.circleParameters.circMode := 1;
   // movePath.pathDataArray[2].commands[9].cmdParameters.circleParameters.circMode := 0;
   // movePath.pathDataArray[2].commands[10].cmdParameters.circleParameters.circMode := 1;
   // movePath.pathDataArray[2].commands[11..20].cmdParameters.circleParameters.circMode := 0;
   // movePath.pathDataArray[3].commands[1..20].cmdParameters.circleParameters.circMode := 0;
   // movePath.pathDataArray[4].commands[1..20].cmdParameters.circleParameters.circMode := 0;
   // movePath.pathDataArray[5].commands[1..20].cmdParameters.circleParameters.circMode := 0;
   // movePath.pathDataArray[1].commands[1..20].cmdParameters.circleParameters.point := -1;
   // movePath.pathDataArray[2].commands[1..20].cmdParameters.circleParameters.point := -1;
   // movePath.pathDataArray[3].commands[1..20].cmdParameters.circleParameters.point := -1;
   // movePath.pathDataArray[4].commands[1..20].cmdParameters.circleParameters.point := -1;
   // movePath.pathDataArray[5].commands[1..20].cmdParameters.circleParameters.point := -1;
   // movePath.pathDataArray[1].commands[1].cmdParameters.circleParameters.auxPoint[1..3] := 0.0;
   // movePath.pathDataArray[1].commands[2].cmdParameters.circleParameters.auxPoint[1..3] := 0.0;
   // movePath.pathDataArray[1].commands[3].cmdParameters.circleParameters.auxPoint[1..3] := 0.0;
   // movePath.pathDataArray[1].commands[4].cmdParameters.circleParameters.auxPoint[1..3] := 0.0;
   // movePath.pathDataArray[1].commands[5].cmdParameters.circleParameters.auxPoint[1..3] := 0.0;
   // movePath.pathDataArray[1].commands[6].cmdParameters.circleParameters.auxPoint[1..3] := 0.0;
   // movePath.pathDataArray[1].commands[7].cmdParameters.circleParameters.auxPoint[1] := 0.0;
   // movePath.pathDataArray[1].commands[7].cmdParameters.circleParameters.auxPoint[2] := 10.0;
   // movePath.pathDataArray[1].commands[7].cmdParameters.circleParameters.auxPoint[3] := 0.0;
   // movePath.pathDataArray[1].commands[8].cmdParameters.circleParameters.auxPoint[1..3] := 0.0;
   // movePath.pathDataArray[1].commands[9].cmdParameters.circleParameters.auxPoint[1] := 0.0;
   // movePath.pathDataArray[1].commands[9].cmdParameters.circleParameters.auxPoint[2] := -10.0;
   // movePath.pathDataArray[1].commands[9].cmdParameters.circleParameters.auxPoint[3] := 0.0;
   // movePath.pathDataArray[1].commands[10].cmdParameters.circleParameters.auxPoint[1..3] := 0.0;
   // movePath.pathDataArray[1].commands[11].cmdParameters.circleParameters.auxPoint[1..3] := 0.0;
   // movePath.pathDataArray[1].commands[12].cmdParameters.circleParameters.auxPoint[1..3] := 0.0;
   // movePath.pathDataArray[1].commands[13].cmdParameters.circleParameters.auxPoint[1..3] := 0.0;
   // movePath.pathDataArray[1].commands[14].cmdParameters.circleParameters.auxPoint[1..3] := 0.0;
   // movePath.pathDataArray[1].commands[15].cmdParameters.circleParameters.auxPoint[1..3] := 0.0;
   // movePath.pathDataArray[1].commands[16].cmdParameters.circleParameters.auxPoint[1..3] := 0.0;
   // movePath.pathDataArray[1].commands[17].cmdParameters.circleParameters.auxPoint[1..3] := 0.0;
   // movePath.pathDataArray[1].commands[18].cmdParameters.circleParameters.auxPoint[1..3] := 0.0;
   // movePath.pathDataArray[1].commands[19].cmdParameters.circleParameters.auxPoint[1..3] := 0.0;
   // movePath.pathDataArray[1].commands[20].cmdParameters.circleParameters.auxPoint[1..3] := 0.0;
   // movePath.pathDataArray[2].commands[1].cmdParameters.circleParameters.auxPoint[1..3] := 0.0;
   // movePath.pathDataArray[2].commands[2].cmdParameters.circleParameters.auxPoint[1..3] := 0.0;
   // movePath.pathDataArray[2].commands[3].cmdParameters.circleParameters.auxPoint[1..3] := 0.0;
   // movePath.pathDataArray[2].commands[4].cmdParameters.circleParameters.auxPoint[1..3] := 0.0;
   // movePath.pathDataArray[2].commands[5].cmdParameters.circleParameters.auxPoint[1..3] := 0.0;
   // movePath.pathDataArray[2].commands[6].cmdParameters.circleParameters.auxPoint[1..3] := 0.0;
   // movePath.pathDataArray[2].commands[7].cmdParameters.circleParameters.auxPoint[1..3] := 0.0;
   // movePath.pathDataArray[2].commands[8].cmdParameters.circleParameters.auxPoint[1] := 0.0;
   // movePath.pathDataArray[2].commands[8].cmdParameters.circleParameters.auxPoint[2] := 10.0;
   // movePath.pathDataArray[2].commands[8].cmdParameters.circleParameters.auxPoint[3] := 0.0;
   // movePath.pathDataArray[2].commands[9].cmdParameters.circleParameters.auxPoint[1..3] := 0.0;
   // movePath.pathDataArray[2].commands[10].cmdParameters.circleParameters.auxPoint[1] := 0.0;
   // movePath.pathDataArray[2].commands[10].cmdParameters.circleParameters.auxPoint[2] := -10.0;
   // movePath.pathDataArray[2].commands[10].cmdParameters.circleParameters.auxPoint[3] := 0.0;
   // movePath.pathDataArray[2].commands[11].cmdParameters.circleParameters.auxPoint[1..3] := 0.0;
   // movePath.pathDataArray[2].commands[12].cmdParameters.circleParameters.auxPoint[1..3] := 0.0;
   // movePath.pathDataArray[2].commands[13].cmdParameters.circleParameters.auxPoint[1..3] := 0.0;
   // movePath.pathDataArray[2].commands[14].cmdParameters.circleParameters.auxPoint[1..3] := 0.0;
   // movePath.pathDataArray[2].commands[15].cmdParameters.circleParameters.auxPoint[1..3] := 0.0;
   // movePath.pathDataArray[2].commands[16].cmdParameters.circleParameters.auxPoint[1..3] := 0.0;
   // movePath.pathDataArray[2].commands[17].cmdParameters.circleParameters.auxPoint[1..3] := 0.0;
   // movePath.pathDataArray[2].commands[18].cmdParameters.circleParameters.auxPoint[1..3] := 0.0;
   // movePath.pathDataArray[2].commands[19].cmdParameters.circleParameters.auxPoint[1..3] := 0.0;
   // movePath.pathDataArray[2].commands[20].cmdParameters.circleParameters.auxPoint[1..3] := 0.0;
   // movePath.pathDataArray[3].commands[1].cmdParameters.circleParameters.auxPoint[1..3] := 0.0;
   // movePath.pathDataArray[3].commands[2].cmdParameters.circleParameters.auxPoint[1..3] := 0.0;
   // movePath.pathDataArray[3].commands[3].cmdParameters.circleParameters.auxPoint[1..3] := 0.0;
   // movePath.pathDataArray[3].commands[4].cmdParameters.circleParameters.auxPoint[1..3] := 0.0;
   // movePath.pathDataArray[3].commands[5].cmdParameters.circleParameters.auxPoint[1..3] := 0.0;
   // movePath.pathDataArray[3].commands[6].cmdParameters.circleParameters.auxPoint[1..3] := 0.0;
   // movePath.pathDataArray[3].commands[7].cmdParameters.circleParameters.auxPoint[1..3] := 0.0;
   // movePath.pathDataArray[3].commands[8].cmdParameters.circleParameters.auxPoint[1..3] := 0.0;
   // movePath.pathDataArray[3].commands[9].cmdParameters.circleParameters.auxPoint[1..3] := 0.0;
   // movePath.pathDataArray[3].commands[10].cmdParameters.circleParameters.auxPoint[1..3] := 0.0;
   // movePath.pathDataArray[3].commands[11].cmdParameters.circleParameters.auxPoint[1..3] := 0.0;
   // movePath.pathDataArray[3].commands[12].cmdParameters.circleParameters.auxPoint[1..3] := 0.0;
   // movePath.pathDataArray[3].commands[13].cmdParameters.circleParameters.auxPoint[1..3] := 0.0;
   // movePath.pathDataArray[3].commands[14].cmdParameters.circleParameters.auxPoint[1..3] := 0.0;
   // movePath.pathDataArray[3].commands[15].cmdParameters.circleParameters.auxPoint[1..3] := 0.0;
   // movePath.pathDataArray[3].commands[16].cmdParameters.circleParameters.auxPoint[1..3] := 0.0;
   // movePath.pathDataArray[3].commands[17].cmdParameters.circleParameters.auxPoint[1..3] := 0.0;
   // movePath.pathDataArray[3].commands[18].cmdParameters.circleParameters.auxPoint[1..3] := 0.0;
   // movePath.pathDataArray[3].commands[19].cmdParameters.circleParameters.auxPoint[1..3] := 0.0;
   // movePath.pathDataArray[3].commands[20].cmdParameters.circleParameters.auxPoint[1..3] := 0.0;
   // movePath.pathDataArray[4].commands[1].cmdParameters.circleParameters.auxPoint[1..3] := 0.0;
   // movePath.pathDataArray[4].commands[2].cmdParameters.circleParameters.auxPoint[1..3] := 0.0;
   // movePath.pathDataArray[4].commands[3].cmdParameters.circleParameters.auxPoint[1..3] := 0.0;
   // movePath.pathDataArray[4].commands[4].cmdParameters.circleParameters.auxPoint[1..3] := 0.0;
   // movePath.pathDataArray[4].commands[5].cmdParameters.circleParameters.auxPoint[1..3] := 0.0;
   // movePath.pathDataArray[4].commands[6].cmdParameters.circleParameters.auxPoint[1..3] := 0.0;
   // movePath.pathDataArray[4].commands[7].cmdParameters.circleParameters.auxPoint[1..3] := 0.0;
   // movePath.pathDataArray[4].commands[8].cmdParameters.circleParameters.auxPoint[1..3] := 0.0;
   // movePath.pathDataArray[4].commands[9].cmdParameters.circleParameters.auxPoint[1..3] := 0.0;
   // movePath.pathDataArray[4].commands[10].cmdParameters.circleParameters.auxPoint[1..3] := 0.0;
   // movePath.pathDataArray[4].commands[11].cmdParameters.circleParameters.auxPoint[1..3] := 0.0;
   // movePath.pathDataArray[4].commands[12].cmdParameters.circleParameters.auxPoint[1..3] := 0.0;
   // movePath.pathDataArray[4].commands[13].cmdParameters.circleParameters.auxPoint[1..3] := 0.0;
   // movePath.pathDataArray[4].commands[14].cmdParameters.circleParameters.auxPoint[1..3] := 0.0;
   // movePath.pathDataArray[4].commands[15].cmdParameters.circleParameters.auxPoint[1..3] := 0.0;
   // movePath.pathDataArray[4].commands[16].cmdParameters.circleParameters.auxPoint[1..3] := 0.0;
   // movePath.pathDataArray[4].commands[17].cmdParameters.circleParameters.auxPoint[1..3] := 0.0;
   // movePath.pathDataArray[4].commands[18].cmdParameters.circleParameters.auxPoint[1..3] := 0.0;
   // movePath.pathDataArray[4].commands[19].cmdParameters.circleParameters.auxPoint[1..3] := 0.0;
   // movePath.pathDataArray[4].commands[20].cmdParameters.circleParameters.auxPoint[1..3] := 0.0;
   // movePath.pathDataArray[5].commands[1].cmdParameters.circleParameters.auxPoint[1..3] := 0.0;
   // movePath.pathDataArray[5].commands[2].cmdParameters.circleParameters.auxPoint[1..3] := 0.0;
   // movePath.pathDataArray[5].commands[3].cmdParameters.circleParameters.auxPoint[1..3] := 0.0;
   // movePath.pathDataArray[5].commands[4].cmdParameters.circleParameters.auxPoint[1..3] := 0.0;
   // movePath.pathDataArray[5].commands[5].cmdParameters.circleParameters.auxPoint[1..3] := 0.0;
   // movePath.pathDataArray[5].commands[6].cmdParameters.circleParameters.auxPoint[1..3] := 0.0;
   // movePath.pathDataArray[5].commands[7].cmdParameters.circleParameters.auxPoint[1..3] := 0.0;
   // movePath.pathDataArray[5].commands[8].cmdParameters.circleParameters.auxPoint[1..3] := 0.0;
   // movePath.pathDataArray[5].commands[9].cmdParameters.circleParameters.auxPoint[1..3] := 0.0;
   // movePath.pathDataArray[5].commands[10].cmdParameters.circleParameters.auxPoint[1..3] := 0.0;
   // movePath.pathDataArray[5].commands[11].cmdParameters.circleParameters.auxPoint[1..3] := 0.0;
   // movePath.pathDataArray[5].commands[12].cmdParameters.circleParameters.auxPoint[1..3] := 0.0;
   // movePath.pathDataArray[5].commands[13].cmdParameters.circleParameters.auxPoint[1..3] := 0.0;
   // movePath.pathDataArray[5].commands[14].cmdParameters.circleParameters.auxPoint[1..3] := 0.0;
   // movePath.pathDataArray[5].commands[15].cmdParameters.circleParameters.auxPoint[1..3] := 0.0;
   // movePath.pathDataArray[5].commands[16].cmdParameters.circleParameters.auxPoint[1..3] := 0.0;
   // movePath.pathDataArray[5].commands[17].cmdParameters.circleParameters.auxPoint[1..3] := 0.0;
   // movePath.pathDataArray[5].commands[18].cmdParameters.circleParameters.auxPoint[1..3] := 0.0;
   // movePath.pathDataArray[5].commands[19].cmdParameters.circleParameters.auxPoint[1..3] := 0.0;
   // movePath.pathDataArray[5].commands[20].cmdParameters.circleParameters.auxPoint[1..3] := 0.0;
   // movePath.pathDataArray[1].commands[1..8].cmdParameters.circleParameters.pathChoice := 0;
   // movePath.pathDataArray[1].commands[9].cmdParameters.circleParameters.pathChoice := 1;
   // movePath.pathDataArray[1].commands[10..20].cmdParameters.circleParameters.pathChoice := 0;
   // movePath.pathDataArray[2].commands[1..9].cmdParameters.circleParameters.pathChoice := 0;
   // movePath.pathDataArray[2].commands[10].cmdParameters.circleParameters.pathChoice := 1;
   // movePath.pathDataArray[2].commands[11..20].cmdParameters.circleParameters.pathChoice := 0;
   // movePath.pathDataArray[3].commands[1..20].cmdParameters.circleParameters.pathChoice := 0;
   // movePath.pathDataArray[4].commands[1..20].cmdParameters.circleParameters.pathChoice := 0;
   // movePath.pathDataArray[5].commands[1..20].cmdParameters.circleParameters.pathChoice := 0;
   // movePath.pathDataArray[1].commands[1..2].cmdParameters.circleParameters.circlePlane := 0;
   // movePath.pathDataArray[1].commands[3].cmdParameters.circleParameters.circlePlane := 2;
   // movePath.pathDataArray[1].commands[4..6].cmdParameters.circleParameters.circlePlane := 0;
   // movePath.pathDataArray[1].commands[7].cmdParameters.circleParameters.circlePlane := 2;
   // movePath.pathDataArray[1].commands[8].cmdParameters.circleParameters.circlePlane := 0;
   // movePath.pathDataArray[1].commands[9].cmdParameters.circleParameters.circlePlane := 2;
   // movePath.pathDataArray[1].commands[10..20].cmdParameters.circleParameters.circlePlane := 0;
   // movePath.pathDataArray[2].commands[1..3].cmdParameters.circleParameters.circlePlane := 0;
   // movePath.pathDataArray[2].commands[4].cmdParameters.circleParameters.circlePlane := 2;
   // movePath.pathDataArray[2].commands[5..7].cmdParameters.circleParameters.circlePlane := 0;
   // movePath.pathDataArray[2].commands[8].cmdParameters.circleParameters.circlePlane := 2;
   // movePath.pathDataArray[2].commands[9].cmdParameters.circleParameters.circlePlane := 0;
   // movePath.pathDataArray[2].commands[10].cmdParameters.circleParameters.circlePlane := 2;
   // movePath.pathDataArray[2].commands[11..20].cmdParameters.circleParameters.circlePlane := 0;
   // movePath.pathDataArray[3].commands[1..20].cmdParameters.circleParameters.circlePlane := 0;
   // movePath.pathDataArray[4].commands[1..20].cmdParameters.circleParameters.circlePlane := 0;
   // movePath.pathDataArray[5].commands[1..20].cmdParameters.circleParameters.circlePlane := 0;
   // movePath.pathDataArray[1].commands[1..20].cmdParameters.circleParameters.radius := 0.0;
   // movePath.pathDataArray[2].commands[1..20].cmdParameters.circleParameters.radius := 0.0;
   // movePath.pathDataArray[3].commands[1..20].cmdParameters.circleParameters.radius := 0.0;
   // movePath.pathDataArray[4].commands[1..20].cmdParameters.circleParameters.radius := 0.0;
   // movePath.pathDataArray[5].commands[1..20].cmdParameters.circleParameters.radius := 0.0;
   // movePath.pathDataArray[1].commands[1..2].cmdParameters.circleParameters.arc := 0.0;
   // movePath.pathDataArray[1].commands[3].cmdParameters.circleParameters.arc := 360.0;
   // movePath.pathDataArray[1].commands[4..6].cmdParameters.circleParameters.arc := 0.0;
   // movePath.pathDataArray[1].commands[7].cmdParameters.circleParameters.arc := 235.0;
   // movePath.pathDataArray[1].commands[8].cmdParameters.circleParameters.arc := 0.0;
   // movePath.pathDataArray[1].commands[9].cmdParameters.circleParameters.arc := 235.0;
   // movePath.pathDataArray[1].commands[10..20].cmdParameters.circleParameters.arc := 0.0;
   // movePath.pathDataArray[2].commands[1..3].cmdParameters.circleParameters.arc := 0.0;
   // movePath.pathDataArray[2].commands[4].cmdParameters.circleParameters.arc := 360.0;
   // movePath.pathDataArray[2].commands[5..7].cmdParameters.circleParameters.arc := 0.0;
   // movePath.pathDataArray[2].commands[8].cmdParameters.circleParameters.arc := 235.0;
   // movePath.pathDataArray[2].commands[9].cmdParameters.circleParameters.arc := 0.0;
   // movePath.pathDataArray[2].commands[10].cmdParameters.circleParameters.arc := 235.0;
   // movePath.pathDataArray[2].commands[11..20].cmdParameters.circleParameters.arc := 0.0;
   // movePath.pathDataArray[3].commands[1..20].cmdParameters.circleParameters.arc := 0.0;
   // movePath.pathDataArray[4].commands[1..20].cmdParameters.circleParameters.arc := 0.0;
   // movePath.pathDataArray[5].commands[1..20].cmdParameters.circleParameters.arc := 0.0;
   // movePath.pathDataArray[1].commands[1..20].cmdParameters.zoneParameters.zoneConfigurationIndex := 0;
   // movePath.pathDataArray[2].commands[1].cmdParameters.zoneParameters.zoneConfigurationIndex := 1;
   // movePath.pathDataArray[2].commands[2..20].cmdParameters.zoneParameters.zoneConfigurationIndex := 0;
   // movePath.pathDataArray[3].commands[1..20].cmdParameters.zoneParameters.zoneConfigurationIndex := 0;
   // movePath.pathDataArray[4].commands[1..20].cmdParameters.zoneParameters.zoneConfigurationIndex := 0;
   // movePath.pathDataArray[5].commands[1..20].cmdParameters.zoneParameters.zoneConfigurationIndex := 0;
   // movePath.pathDataArray[1].commands[1..20].cmdParameters.zoneParameters.zoneNumber := 0;
   // movePath.pathDataArray[2].commands[1].cmdParameters.zoneParameters.zoneNumber := 1;
   // movePath.pathDataArray[2].commands[2..20].cmdParameters.zoneParameters.zoneNumber := 0;
   // movePath.pathDataArray[3].commands[1..20].cmdParameters.zoneParameters.zoneNumber := 0;
   // movePath.pathDataArray[4].commands[1..20].cmdParameters.zoneParameters.zoneNumber := 0;
   // movePath.pathDataArray[5].commands[1..20].cmdParameters.zoneParameters.zoneNumber := 0;
   // movePath.pathDataArray[1].commands[1..20].cmdParameters.zoneParameters.deactivationMode := 0;
   // movePath.pathDataArray[2].commands[1..20].cmdParameters.zoneParameters.deactivationMode := 0;
   // movePath.pathDataArray[3].commands[1..20].cmdParameters.zoneParameters.deactivationMode := 0;
   // movePath.pathDataArray[4].commands[1..20].cmdParameters.zoneParameters.deactivationMode := 0;
   // movePath.pathDataArray[5].commands[1..20].cmdParameters.zoneParameters.deactivationMode := 0;
   // movePath.pathDataArray[1].commands[1].cmdParameters.pickAndPlaceParameters.startParameter.direction[1..3] := 0.0;
   // movePath.pathDataArray[1].commands[2].cmdParameters.pickAndPlaceParameters.startParameter.direction[1..3] := 0.0;
   // movePath.pathDataArray[1].commands[3].cmdParameters.pickAndPlaceParameters.startParameter.direction[1..3] := 0.0;
   // movePath.pathDataArray[1].commands[4].cmdParameters.pickAndPlaceParameters.startParameter.direction[1..3] := 0.0;
   // movePath.pathDataArray[1].commands[5].cmdParameters.pickAndPlaceParameters.startParameter.direction[1..3] := 0.0;
   // movePath.pathDataArray[1].commands[6].cmdParameters.pickAndPlaceParameters.startParameter.direction[1..3] := 0.0;
   // movePath.pathDataArray[1].commands[7].cmdParameters.pickAndPlaceParameters.startParameter.direction[1..3] := 0.0;
   // movePath.pathDataArray[1].commands[8].cmdParameters.pickAndPlaceParameters.startParameter.direction[1..3] := 0.0;
   // movePath.pathDataArray[1].commands[9].cmdParameters.pickAndPlaceParameters.startParameter.direction[1..3] := 0.0;
   // movePath.pathDataArray[1].commands[10].cmdParameters.pickAndPlaceParameters.startParameter.direction[1..3] := 0.0;
   // movePath.pathDataArray[1].commands[11].cmdParameters.pickAndPlaceParameters.startParameter.direction[1..3] := 0.0;
   // movePath.pathDataArray[1].commands[12].cmdParameters.pickAndPlaceParameters.startParameter.direction[1..3] := 0.0;
   // movePath.pathDataArray[1].commands[13].cmdParameters.pickAndPlaceParameters.startParameter.direction[1..3] := 0.0;
   // movePath.pathDataArray[1].commands[14].cmdParameters.pickAndPlaceParameters.startParameter.direction[1..3] := 0.0;
   // movePath.pathDataArray[1].commands[15].cmdParameters.pickAndPlaceParameters.startParameter.direction[1..3] := 0.0;
   // movePath.pathDataArray[1].commands[16].cmdParameters.pickAndPlaceParameters.startParameter.direction[1..3] := 0.0;
   // movePath.pathDataArray[1].commands[17].cmdParameters.pickAndPlaceParameters.startParameter.direction[1..3] := 0.0;
   // movePath.pathDataArray[1].commands[18].cmdParameters.pickAndPlaceParameters.startParameter.direction[1..3] := 0.0;
   // movePath.pathDataArray[1].commands[19].cmdParameters.pickAndPlaceParameters.startParameter.direction[1..3] := 0.0;
   // movePath.pathDataArray[1].commands[20].cmdParameters.pickAndPlaceParameters.startParameter.direction[1..3] := 0.0;
   // movePath.pathDataArray[2].commands[1].cmdParameters.pickAndPlaceParameters.startParameter.direction[1..3] := 0.0;
   // movePath.pathDataArray[2].commands[2].cmdParameters.pickAndPlaceParameters.startParameter.direction[1..3] := 0.0;
   // movePath.pathDataArray[2].commands[3].cmdParameters.pickAndPlaceParameters.startParameter.direction[1..3] := 0.0;
   // movePath.pathDataArray[2].commands[4].cmdParameters.pickAndPlaceParameters.startParameter.direction[1..3] := 0.0;
   // movePath.pathDataArray[2].commands[5].cmdParameters.pickAndPlaceParameters.startParameter.direction[1..3] := 0.0;
   // movePath.pathDataArray[2].commands[6].cmdParameters.pickAndPlaceParameters.startParameter.direction[1..3] := 0.0;
   // movePath.pathDataArray[2].commands[7].cmdParameters.pickAndPlaceParameters.startParameter.direction[1..3] := 0.0;
   // movePath.pathDataArray[2].commands[8].cmdParameters.pickAndPlaceParameters.startParameter.direction[1..3] := 0.0;
   // movePath.pathDataArray[2].commands[9].cmdParameters.pickAndPlaceParameters.startParameter.direction[1..3] := 0.0;
   // movePath.pathDataArray[2].commands[10].cmdParameters.pickAndPlaceParameters.startParameter.direction[1..3] := 0.0;
   // movePath.pathDataArray[2].commands[11].cmdParameters.pickAndPlaceParameters.startParameter.direction[1..3] := 0.0;
   // movePath.pathDataArray[2].commands[12].cmdParameters.pickAndPlaceParameters.startParameter.direction[1..3] := 0.0;
   // movePath.pathDataArray[2].commands[13].cmdParameters.pickAndPlaceParameters.startParameter.direction[1..3] := 0.0;
   // movePath.pathDataArray[2].commands[14].cmdParameters.pickAndPlaceParameters.startParameter.direction[1..3] := 0.0;
   // movePath.pathDataArray[2].commands[15].cmdParameters.pickAndPlaceParameters.startParameter.direction[1..3] := 0.0;
   // movePath.pathDataArray[2].commands[16].cmdParameters.pickAndPlaceParameters.startParameter.direction[1..3] := 0.0;
   // movePath.pathDataArray[2].commands[17].cmdParameters.pickAndPlaceParameters.startParameter.direction[1..3] := 0.0;
   // movePath.pathDataArray[2].commands[18].cmdParameters.pickAndPlaceParameters.startParameter.direction[1..3] := 0.0;
   // movePath.pathDataArray[2].commands[19].cmdParameters.pickAndPlaceParameters.startParameter.direction[1..3] := 0.0;
   // movePath.pathDataArray[2].commands[20].cmdParameters.pickAndPlaceParameters.startParameter.direction[1..3] := 0.0;
   // movePath.pathDataArray[3].commands[1].cmdParameters.pickAndPlaceParameters.startParameter.direction[1..3] := 0.0;
   // movePath.pathDataArray[3].commands[2].cmdParameters.pickAndPlaceParameters.startParameter.direction[1..3] := 0.0;
   // movePath.pathDataArray[3].commands[3].cmdParameters.pickAndPlaceParameters.startParameter.direction[1..3] := 0.0;
   // movePath.pathDataArray[3].commands[4].cmdParameters.pickAndPlaceParameters.startParameter.direction[1..3] := 0.0;
   // movePath.pathDataArray[3].commands[5].cmdParameters.pickAndPlaceParameters.startParameter.direction[1..3] := 0.0;
   // movePath.pathDataArray[3].commands[6].cmdParameters.pickAndPlaceParameters.startParameter.direction[1..3] := 0.0;
   // movePath.pathDataArray[3].commands[7].cmdParameters.pickAndPlaceParameters.startParameter.direction[1..3] := 0.0;
   // movePath.pathDataArray[3].commands[8].cmdParameters.pickAndPlaceParameters.startParameter.direction[1..3] := 0.0;
   // movePath.pathDataArray[3].commands[9].cmdParameters.pickAndPlaceParameters.startParameter.direction[1..3] := 0.0;
   // movePath.pathDataArray[3].commands[10].cmdParameters.pickAndPlaceParameters.startParameter.direction[1..3] := 0.0;
   // movePath.pathDataArray[3].commands[11].cmdParameters.pickAndPlaceParameters.startParameter.direction[1..3] := 0.0;
   // movePath.pathDataArray[3].commands[12].cmdParameters.pickAndPlaceParameters.startParameter.direction[1..3] := 0.0;
   // movePath.pathDataArray[3].commands[13].cmdParameters.pickAndPlaceParameters.startParameter.direction[1..3] := 0.0;
   // movePath.pathDataArray[3].commands[14].cmdParameters.pickAndPlaceParameters.startParameter.direction[1..3] := 0.0;
   // movePath.pathDataArray[3].commands[15].cmdParameters.pickAndPlaceParameters.startParameter.direction[1..3] := 0.0;
   // movePath.pathDataArray[3].commands[16].cmdParameters.pickAndPlaceParameters.startParameter.direction[1..3] := 0.0;
   // movePath.pathDataArray[3].commands[17].cmdParameters.pickAndPlaceParameters.startParameter.direction[1..3] := 0.0;
   // movePath.pathDataArray[3].commands[18].cmdParameters.pickAndPlaceParameters.startParameter.direction[1..3] := 0.0;
   // movePath.pathDataArray[3].commands[19].cmdParameters.pickAndPlaceParameters.startParameter.direction[1..3] := 0.0;
   // movePath.pathDataArray[3].commands[20].cmdParameters.pickAndPlaceParameters.startParameter.direction[1..3] := 0.0;
   // movePath.pathDataArray[4].commands[1].cmdParameters.pickAndPlaceParameters.startParameter.direction[1..3] := 0.0;
   // movePath.pathDataArray[4].commands[2].cmdParameters.pickAndPlaceParameters.startParameter.direction[1..3] := 0.0;
   // movePath.pathDataArray[4].commands[3].cmdParameters.pickAndPlaceParameters.startParameter.direction[1..3] := 0.0;
   // movePath.pathDataArray[4].commands[4].cmdParameters.pickAndPlaceParameters.startParameter.direction[1..2] := 0.0;
   // movePath.pathDataArray[4].commands[4].cmdParameters.pickAndPlaceParameters.startParameter.direction[3] := 1.0;
   // movePath.pathDataArray[4].commands[5].cmdParameters.pickAndPlaceParameters.startParameter.direction[1..3] := 0.0;
   // movePath.pathDataArray[4].commands[6].cmdParameters.pickAndPlaceParameters.startParameter.direction[1..2] := 0.0;
   // movePath.pathDataArray[4].commands[6].cmdParameters.pickAndPlaceParameters.startParameter.direction[3] := 1.0;
   // movePath.pathDataArray[4].commands[7].cmdParameters.pickAndPlaceParameters.startParameter.direction[1..3] := 0.0;
   // movePath.pathDataArray[4].commands[8].cmdParameters.pickAndPlaceParameters.startParameter.direction[1..3] := 0.0;
   // movePath.pathDataArray[4].commands[9].cmdParameters.pickAndPlaceParameters.startParameter.direction[1..3] := 0.0;
   // movePath.pathDataArray[4].commands[10].cmdParameters.pickAndPlaceParameters.startParameter.direction[1..3] := 0.0;
   // movePath.pathDataArray[4].commands[11].cmdParameters.pickAndPlaceParameters.startParameter.direction[1..3] := 0.0;
   // movePath.pathDataArray[4].commands[12].cmdParameters.pickAndPlaceParameters.startParameter.direction[1..3] := 0.0;
   // movePath.pathDataArray[4].commands[13].cmdParameters.pickAndPlaceParameters.startParameter.direction[1..3] := 0.0;
   // movePath.pathDataArray[4].commands[14].cmdParameters.pickAndPlaceParameters.startParameter.direction[1..3] := 0.0;
   // movePath.pathDataArray[4].commands[15].cmdParameters.pickAndPlaceParameters.startParameter.direction[1..3] := 0.0;
   // movePath.pathDataArray[4].commands[16].cmdParameters.pickAndPlaceParameters.startParameter.direction[1..3] := 0.0;
   // movePath.pathDataArray[4].commands[17].cmdParameters.pickAndPlaceParameters.startParameter.direction[1..3] := 0.0;
   // movePath.pathDataArray[4].commands[18].cmdParameters.pickAndPlaceParameters.startParameter.direction[1..3] := 0.0;
   // movePath.pathDataArray[4].commands[19].cmdParameters.pickAndPlaceParameters.startParameter.direction[1..3] := 0.0;
   // movePath.pathDataArray[4].commands[20].cmdParameters.pickAndPlaceParameters.startParameter.direction[1..3] := 0.0;
   // movePath.pathDataArray[5].commands[1].cmdParameters.pickAndPlaceParameters.startParameter.direction[1..3] := 0.0;
   // movePath.pathDataArray[5].commands[2].cmdParameters.pickAndPlaceParameters.startParameter.direction[1..3] := 0.0;
   // movePath.pathDataArray[5].commands[3].cmdParameters.pickAndPlaceParameters.startParameter.direction[1..3] := 0.0;
   // movePath.pathDataArray[5].commands[4].cmdParameters.pickAndPlaceParameters.startParameter.direction[1..3] := 0.0;
   // movePath.pathDataArray[5].commands[5].cmdParameters.pickAndPlaceParameters.startParameter.direction[1..3] := 0.0;
   // movePath.pathDataArray[5].commands[6].cmdParameters.pickAndPlaceParameters.startParameter.direction[1..3] := 0.0;
   // movePath.pathDataArray[5].commands[7].cmdParameters.pickAndPlaceParameters.startParameter.direction[1..3] := 0.0;
   // movePath.pathDataArray[5].commands[8].cmdParameters.pickAndPlaceParameters.startParameter.direction[1..3] := 0.0;
   // movePath.pathDataArray[5].commands[9].cmdParameters.pickAndPlaceParameters.startParameter.direction[1..3] := 0.0;
   // movePath.pathDataArray[5].commands[10].cmdParameters.pickAndPlaceParameters.startParameter.direction[1..3] := 0.0;
   // movePath.pathDataArray[5].commands[11].cmdParameters.pickAndPlaceParameters.startParameter.direction[1..3] := 0.0;
   // movePath.pathDataArray[5].commands[12].cmdParameters.pickAndPlaceParameters.startParameter.direction[1..3] := 0.0;
   // movePath.pathDataArray[5].commands[13].cmdParameters.pickAndPlaceParameters.startParameter.direction[1..3] := 0.0;
   // movePath.pathDataArray[5].commands[14].cmdParameters.pickAndPlaceParameters.startParameter.direction[1..3] := 0.0;
   // movePath.pathDataArray[5].commands[15].cmdParameters.pickAndPlaceParameters.startParameter.direction[1..3] := 0.0;
   // movePath.pathDataArray[5].commands[16].cmdParameters.pickAndPlaceParameters.startParameter.direction[1..3] := 0.0;
   // movePath.pathDataArray[5].commands[17].cmdParameters.pickAndPlaceParameters.startParameter.direction[1..3] := 0.0;
   // movePath.pathDataArray[5].commands[18].cmdParameters.pickAndPlaceParameters.startParameter.direction[1..3] := 0.0;
   // movePath.pathDataArray[5].commands[19].cmdParameters.pickAndPlaceParameters.startParameter.direction[1..3] := 0.0;
   // movePath.pathDataArray[5].commands[20].cmdParameters.pickAndPlaceParameters.startParameter.direction[1..3] := 0.0;
   // movePath.pathDataArray[1].commands[1..20].cmdParameters.pickAndPlaceParameters.startParameter.workingHeight := 0.0;
   // movePath.pathDataArray[2].commands[1..20].cmdParameters.pickAndPlaceParameters.startParameter.workingHeight := 0.0;
   // movePath.pathDataArray[3].commands[1..20].cmdParameters.pickAndPlaceParameters.startParameter.workingHeight := 0.0;
   // movePath.pathDataArray[4].commands[1..3].cmdParameters.pickAndPlaceParameters.startParameter.workingHeight := 0.0;
   // movePath.pathDataArray[4].commands[4].cmdParameters.pickAndPlaceParameters.startParameter.workingHeight := 60.0;
   // movePath.pathDataArray[4].commands[5].cmdParameters.pickAndPlaceParameters.startParameter.workingHeight := 0.0;
   // movePath.pathDataArray[4].commands[6].cmdParameters.pickAndPlaceParameters.startParameter.workingHeight := 60.0;
   // movePath.pathDataArray[4].commands[7..20].cmdParameters.pickAndPlaceParameters.startParameter.workingHeight := 0.0;
   // movePath.pathDataArray[5].commands[1..20].cmdParameters.pickAndPlaceParameters.startParameter.workingHeight := 0.0;
   // movePath.pathDataArray[1].commands[1..20].cmdParameters.pickAndPlaceParameters.startParameter.transitionArea := 0.0;
   // movePath.pathDataArray[2].commands[1..20].cmdParameters.pickAndPlaceParameters.startParameter.transitionArea := 0.0;
   // movePath.pathDataArray[3].commands[1..20].cmdParameters.pickAndPlaceParameters.startParameter.transitionArea := 0.0;
   // movePath.pathDataArray[4].commands[1..20].cmdParameters.pickAndPlaceParameters.startParameter.transitionArea := 0.0;
   // movePath.pathDataArray[5].commands[1..20].cmdParameters.pickAndPlaceParameters.startParameter.transitionArea := 0.0;
   // movePath.pathDataArray[1].commands[1..20].cmdParameters.pickAndPlaceParameters.startParameter.dynamicsFactor := 100.0;
   // movePath.pathDataArray[2].commands[1..20].cmdParameters.pickAndPlaceParameters.startParameter.dynamicsFactor := 100.0;
   // movePath.pathDataArray[3].commands[1..20].cmdParameters.pickAndPlaceParameters.startParameter.dynamicsFactor := 100.0;
   // movePath.pathDataArray[4].commands[1..20].cmdParameters.pickAndPlaceParameters.startParameter.dynamicsFactor := 100.0;
   // movePath.pathDataArray[5].commands[1..20].cmdParameters.pickAndPlaceParameters.startParameter.dynamicsFactor := 100.0;
   // movePath.pathDataArray[1].commands[1].cmdParameters.pickAndPlaceParameters.targetParameter.direction[1..3] := 0.0;
   // movePath.pathDataArray[1].commands[2].cmdParameters.pickAndPlaceParameters.targetParameter.direction[1..3] := 0.0;
   // movePath.pathDataArray[1].commands[3].cmdParameters.pickAndPlaceParameters.targetParameter.direction[1..3] := 0.0;
   // movePath.pathDataArray[1].commands[4].cmdParameters.pickAndPlaceParameters.targetParameter.direction[1..3] := 0.0;
   // movePath.pathDataArray[1].commands[5].cmdParameters.pickAndPlaceParameters.targetParameter.direction[1..3] := 0.0;
   // movePath.pathDataArray[1].commands[6].cmdParameters.pickAndPlaceParameters.targetParameter.direction[1..3] := 0.0;
   // movePath.pathDataArray[1].commands[7].cmdParameters.pickAndPlaceParameters.targetParameter.direction[1..3] := 0.0;
   // movePath.pathDataArray[1].commands[8].cmdParameters.pickAndPlaceParameters.targetParameter.direction[1..3] := 0.0;
   // movePath.pathDataArray[1].commands[9].cmdParameters.pickAndPlaceParameters.targetParameter.direction[1..3] := 0.0;
   // movePath.pathDataArray[1].commands[10].cmdParameters.pickAndPlaceParameters.targetParameter.direction[1..3] := 0.0;
   // movePath.pathDataArray[1].commands[11].cmdParameters.pickAndPlaceParameters.targetParameter.direction[1..3] := 0.0;
   // movePath.pathDataArray[1].commands[12].cmdParameters.pickAndPlaceParameters.targetParameter.direction[1..3] := 0.0;
   // movePath.pathDataArray[1].commands[13].cmdParameters.pickAndPlaceParameters.targetParameter.direction[1..3] := 0.0;
   // movePath.pathDataArray[1].commands[14].cmdParameters.pickAndPlaceParameters.targetParameter.direction[1..3] := 0.0;
   // movePath.pathDataArray[1].commands[15].cmdParameters.pickAndPlaceParameters.targetParameter.direction[1..3] := 0.0;
   // movePath.pathDataArray[1].commands[16].cmdParameters.pickAndPlaceParameters.targetParameter.direction[1..3] := 0.0;
   // movePath.pathDataArray[1].commands[17].cmdParameters.pickAndPlaceParameters.targetParameter.direction[1..3] := 0.0;
   // movePath.pathDataArray[1].commands[18].cmdParameters.pickAndPlaceParameters.targetParameter.direction[1..3] := 0.0;
   // movePath.pathDataArray[1].commands[19].cmdParameters.pickAndPlaceParameters.targetParameter.direction[1..3] := 0.0;
   // movePath.pathDataArray[1].commands[20].cmdParameters.pickAndPlaceParameters.targetParameter.direction[1..3] := 0.0;
   // movePath.pathDataArray[2].commands[1].cmdParameters.pickAndPlaceParameters.targetParameter.direction[1..3] := 0.0;
   // movePath.pathDataArray[2].commands[2].cmdParameters.pickAndPlaceParameters.targetParameter.direction[1..3] := 0.0;
   // movePath.pathDataArray[2].commands[3].cmdParameters.pickAndPlaceParameters.targetParameter.direction[1..3] := 0.0;
   // movePath.pathDataArray[2].commands[4].cmdParameters.pickAndPlaceParameters.targetParameter.direction[1..3] := 0.0;
   // movePath.pathDataArray[2].commands[5].cmdParameters.pickAndPlaceParameters.targetParameter.direction[1..3] := 0.0;
   // movePath.pathDataArray[2].commands[6].cmdParameters.pickAndPlaceParameters.targetParameter.direction[1..3] := 0.0;
   // movePath.pathDataArray[2].commands[7].cmdParameters.pickAndPlaceParameters.targetParameter.direction[1..3] := 0.0;
   // movePath.pathDataArray[2].commands[8].cmdParameters.pickAndPlaceParameters.targetParameter.direction[1..3] := 0.0;
   // movePath.pathDataArray[2].commands[9].cmdParameters.pickAndPlaceParameters.targetParameter.direction[1..3] := 0.0;
   // movePath.pathDataArray[2].commands[10].cmdParameters.pickAndPlaceParameters.targetParameter.direction[1..3] := 0.0;
   // movePath.pathDataArray[2].commands[11].cmdParameters.pickAndPlaceParameters.targetParameter.direction[1..3] := 0.0;
   // movePath.pathDataArray[2].commands[12].cmdParameters.pickAndPlaceParameters.targetParameter.direction[1..3] := 0.0;
   // movePath.pathDataArray[2].commands[13].cmdParameters.pickAndPlaceParameters.targetParameter.direction[1..3] := 0.0;
   // movePath.pathDataArray[2].commands[14].cmdParameters.pickAndPlaceParameters.targetParameter.direction[1..3] := 0.0;
   // movePath.pathDataArray[2].commands[15].cmdParameters.pickAndPlaceParameters.targetParameter.direction[1..3] := 0.0;
   // movePath.pathDataArray[2].commands[16].cmdParameters.pickAndPlaceParameters.targetParameter.direction[1..3] := 0.0;
   // movePath.pathDataArray[2].commands[17].cmdParameters.pickAndPlaceParameters.targetParameter.direction[1..3] := 0.0;
   // movePath.pathDataArray[2].commands[18].cmdParameters.pickAndPlaceParameters.targetParameter.direction[1..3] := 0.0;
   // movePath.pathDataArray[2].commands[19].cmdParameters.pickAndPlaceParameters.targetParameter.direction[1..3] := 0.0;
   // movePath.pathDataArray[2].commands[20].cmdParameters.pickAndPlaceParameters.targetParameter.direction[1..3] := 0.0;
   // movePath.pathDataArray[3].commands[1].cmdParameters.pickAndPlaceParameters.targetParameter.direction[1..3] := 0.0;
   // movePath.pathDataArray[3].commands[2].cmdParameters.pickAndPlaceParameters.targetParameter.direction[1..3] := 0.0;
   // movePath.pathDataArray[3].commands[3].cmdParameters.pickAndPlaceParameters.targetParameter.direction[1..3] := 0.0;
   // movePath.pathDataArray[3].commands[4].cmdParameters.pickAndPlaceParameters.targetParameter.direction[1..3] := 0.0;
   // movePath.pathDataArray[3].commands[5].cmdParameters.pickAndPlaceParameters.targetParameter.direction[1..3] := 0.0;
   // movePath.pathDataArray[3].commands[6].cmdParameters.pickAndPlaceParameters.targetParameter.direction[1..3] := 0.0;
   // movePath.pathDataArray[3].commands[7].cmdParameters.pickAndPlaceParameters.targetParameter.direction[1..3] := 0.0;
   // movePath.pathDataArray[3].commands[8].cmdParameters.pickAndPlaceParameters.targetParameter.direction[1..3] := 0.0;
   // movePath.pathDataArray[3].commands[9].cmdParameters.pickAndPlaceParameters.targetParameter.direction[1..3] := 0.0;
   // movePath.pathDataArray[3].commands[10].cmdParameters.pickAndPlaceParameters.targetParameter.direction[1..3] := 0.0;
   // movePath.pathDataArray[3].commands[11].cmdParameters.pickAndPlaceParameters.targetParameter.direction[1..3] := 0.0;
   // movePath.pathDataArray[3].commands[12].cmdParameters.pickAndPlaceParameters.targetParameter.direction[1..3] := 0.0;
   // movePath.pathDataArray[3].commands[13].cmdParameters.pickAndPlaceParameters.targetParameter.direction[1..3] := 0.0;
   // movePath.pathDataArray[3].commands[14].cmdParameters.pickAndPlaceParameters.targetParameter.direction[1..3] := 0.0;
   // movePath.pathDataArray[3].commands[15].cmdParameters.pickAndPlaceParameters.targetParameter.direction[1..3] := 0.0;
   // movePath.pathDataArray[3].commands[16].cmdParameters.pickAndPlaceParameters.targetParameter.direction[1..3] := 0.0;
   // movePath.pathDataArray[3].commands[17].cmdParameters.pickAndPlaceParameters.targetParameter.direction[1..3] := 0.0;
   // movePath.pathDataArray[3].commands[18].cmdParameters.pickAndPlaceParameters.targetParameter.direction[1..3] := 0.0;
   // movePath.pathDataArray[3].commands[19].cmdParameters.pickAndPlaceParameters.targetParameter.direction[1..3] := 0.0;
   // movePath.pathDataArray[3].commands[20].cmdParameters.pickAndPlaceParameters.targetParameter.direction[1..3] := 0.0;
   // movePath.pathDataArray[4].commands[1].cmdParameters.pickAndPlaceParameters.targetParameter.direction[1..3] := 0.0;
   // movePath.pathDataArray[4].commands[2].cmdParameters.pickAndPlaceParameters.targetParameter.direction[1..2] := 0.0;
   // movePath.pathDataArray[4].commands[2].cmdParameters.pickAndPlaceParameters.targetParameter.direction[3] := 1.0;
   // movePath.pathDataArray[4].commands[3].cmdParameters.pickAndPlaceParameters.targetParameter.direction[1..3] := 0.0;
   // movePath.pathDataArray[4].commands[4].cmdParameters.pickAndPlaceParameters.targetParameter.direction[1..2] := 0.0;
   // movePath.pathDataArray[4].commands[4].cmdParameters.pickAndPlaceParameters.targetParameter.direction[3] := 1.0;
   // movePath.pathDataArray[4].commands[5].cmdParameters.pickAndPlaceParameters.targetParameter.direction[1..3] := 0.0;
   // movePath.pathDataArray[4].commands[6].cmdParameters.pickAndPlaceParameters.targetParameter.direction[1..3] := 0.0;
   // movePath.pathDataArray[4].commands[7].cmdParameters.pickAndPlaceParameters.targetParameter.direction[1..3] := 0.0;
   // movePath.pathDataArray[4].commands[8].cmdParameters.pickAndPlaceParameters.targetParameter.direction[1..3] := 0.0;
   // movePath.pathDataArray[4].commands[9].cmdParameters.pickAndPlaceParameters.targetParameter.direction[1..3] := 0.0;
   // movePath.pathDataArray[4].commands[10].cmdParameters.pickAndPlaceParameters.targetParameter.direction[1..3] := 0.0;
   // movePath.pathDataArray[4].commands[11].cmdParameters.pickAndPlaceParameters.targetParameter.direction[1..3] := 0.0;
   // movePath.pathDataArray[4].commands[12].cmdParameters.pickAndPlaceParameters.targetParameter.direction[1..3] := 0.0;
   // movePath.pathDataArray[4].commands[13].cmdParameters.pickAndPlaceParameters.targetParameter.direction[1..3] := 0.0;
   // movePath.pathDataArray[4].commands[14].cmdParameters.pickAndPlaceParameters.targetParameter.direction[1..3] := 0.0;
   // movePath.pathDataArray[4].commands[15].cmdParameters.pickAndPlaceParameters.targetParameter.direction[1..3] := 0.0;
   // movePath.pathDataArray[4].commands[16].cmdParameters.pickAndPlaceParameters.targetParameter.direction[1..3] := 0.0;
